// TIA Portal project "Njegovec_diplomski_PLC_HMI" (V19)

(* hardware
DEVICE "S7-1500/ET200MP station_1"  S7-1500 station
   slot 0: "Rail_0"  Rack  6ES7 590-1***0-0AA0
   slot 1: "PLC_1"  CPU 1513-1 PN  6ES7 513-1AL02-0AB0  V2.6
      slot 3: "CPU display_1"  6ES7591-1AA00-0AA0
      slot 32768: "PROFINET interface_1"  X1
DEVICE "HMI_1"  KTP700 Basic PN
   slot 0: "HMI_1"  KTP700 Basic PN  6AV2 123-2GB03-0AX0  17.0.0.0
   slot 1: "HMI_RT_1"  KTP700 Basic PN  6AV2 123-2GB03-0AX0  17.0.0.0
   slot 5: "HMI_1.IE_CP_1"  PROFINET Interface  17.0.0.0
      slot 1: "PROFINET Interface_1"  PROFINET Interface
         slot 1: "Port_1"  Port
*)

// ===== PLC "PLC_1"  CPU 1513-1 PN =====

VAR_GLOBAL   // PLC tag table "Default tag table"
   "air_ON" AT %M4.0 : Bool;
   "System_Byte" AT %MB100 : Byte;
   "FirstScan" AT %M100.0 : Bool;
   "DiagStatusUpdate" AT %M100.1 : Bool;
   "AlwaysTRUE" AT %M100.2 : Bool;
   "AlwaysFALSE" AT %M100.3 : Bool;
   "Clock_Byte" AT %MB105 : Byte;
   "Clock_10Hz" AT %M105.0 : Bool;
   "Clock_5Hz" AT %M105.1 : Bool;
   "Clock_2.5Hz" AT %M105.2 : Bool;
   "Clock_2Hz" AT %M105.3 : Bool;
   "Clock_1.25Hz" AT %M105.4 : Bool;
   "Clock_1Hz" AT %M105.5 : Bool;
   "Clock_0.625Hz" AT %M105.6 : Bool;
   "Clock_0.5Hz" AT %M105.7 : Bool;
END_VAR

VAR_GLOBAL   // PLC tag table "Okretni stol"
   "ventil_1_ukljuci" AT %Q0.1 : Bool;
   "ventil_1_iskljuci" AT %Q0.2 : Bool;
   "stol_okret" AT %Q1.5 : Bool;
   "ventil_2_ukljuci" AT %Q0.3 : Bool;
   "ventil_2_iskljuci" AT %Q0.4 : Bool;
   "clamp_1_1_otvoren" AT %I0.1 : Bool;
   "clamp_2_1_otvoren" AT %I0.3 : Bool;
   "clamp_3_1_otvoren" AT %I0.5 : Bool;
   "clamp_4_1_otvoren" AT %I0.7 : Bool;
   "clamp_5_1_otvoren" AT %I1.1 : Bool;
   "clamp_1_2_otvoren" AT %I1.3 : Bool;
   "clamp_2_2_otvoren" AT %I1.5 : Bool;
   "clamp_3_2_otvoren" AT %I1.7 : Bool;
   "clamp_4_2_otvoren" AT %I2.1 : Bool;
   "clamp_5_2_otvoren" AT %I2.3 : Bool;
   "pin_1_1_izvucen" AT %I2.5 : Bool;
   "pin_2_1_izvucen" AT %I2.7 : Bool;
   "pin_3_1_izvucen" AT %I3.1 : Bool;
   "pin_1_2_izvucen" AT %I3.3 : Bool;
   "pin_2_2_izvucen" AT %I3.5 : Bool;
   "pin_3_2_izvucen" AT %I3.7 : Bool;
   "clamp_1_1_zatvoren" AT %I0.0 : Bool;
   "clamp_2_1_zatvoren" AT %I0.2 : Bool;
   "clamp_3_1_zatvoren" AT %I0.4 : Bool;
   "clamp_4_1_zatvoren" AT %I0.6 : Bool;
   "clamp_5_1_zatvoren" AT %I1.0 : Bool;
   "clamp_1_2_zatvoren" AT %I1.2 : Bool;
   "clamp_2_2_zatvoren" AT %I1.4 : Bool;
   "clamp_3_2_zatvoren" AT %I1.6 : Bool;
   "clamp_4_2_zatvoren" AT %I2.0 : Bool;
   "clamp_5_2_zatvoren" AT %I2.2 : Bool;
   "pin_1_1_uvucen" AT %I2.4 : Bool;
   "pin_2_1_uvucen" AT %I2.6 : Bool;
   "pin_3_1_uvucen" AT %I3.0 : Bool;
   "pin_1_2_uvucen" AT %I3.2 : Bool;
   "pin_2_2_uvucen" AT %I3.4 : Bool;
   "pin_3_2_uvucen" AT %I3.6 : Bool;
   "ventil_pin_1_uklj" AT %Q1.1 : Bool;
   "ventil_pin_1_isklj" AT %Q1.2 : Bool;
   "ventil_pin_2_uklj" AT %Q1.3 : Bool;
   "ventil_pin_2_isklj" AT %Q1.4 : Bool;
   "stol_povratak" AT %Q1.6 : Bool;
   "stol_home" AT %I4.0 : Bool;
   "stol_final" AT %I4.1 : Bool;
END_VAR

VAR_GLOBAL   // PLC tag table "Tipkalo"
   "zeleno" AT %M1.0 : Bool;
   "bijelo" AT %M1.1 : Bool;
   "plavo" AT %M1.2 : Bool;
   "zahtjev_vrata" AT %M1.3 : Bool;
END_VAR

VAR_GLOBAL   // PLC tag table "Robot"
   "robot_move_enable" AT %M2.0 : Bool;
   "KR120_R2700_2_at_HOME" AT %I5.0 : Bool;
   "KR120_R2700_2_startProgram" AT %Q2.0 : Bool;
   "KR120_R2700_2_emergencyStop" AT %Q2.1 : Bool;
   "KR120_R2700_2_programPause" AT %Q2.2 : Bool;
   "KR120_R2700_2_programEnded" AT %I5.1 : Bool;
   "KR120_R2700_2_robotReady" AT %I5.2 : Bool;
   "KR120_R2700_2_mirrorProgramNumber" AT %IB6 : Byte;
   "KR120_R2700_2_programNumber" AT %QB6 : Byte;
   "Zavar_gotov" AT %I8.6 : Bool;
   "handshake_test_out" AT %Q4.0 : Bool;
   "pocetak_rada" AT %I7.1 : Bool;
END_VAR

VAR_GLOBAL   // PLC tag table "Safety"
   "EstopOK" AT %M3.0 : Bool;
END_VAR

VAR_GLOBAL   // PLC tag table "Vrata"
   "vrata_otvori" AT %Q3.0 : Bool;
   "vrata_zatvori" AT %Q3.1 : Bool;
   "lock_zat" AT %Q4.1 : Bool;
   "lock_otv" AT %Q4.2 : Bool;
   "otvoren_lock" AT %I7.0 : Bool;
   "zatvoren_lock" AT %I7.2 : Bool;
   "rolo_vrata_zatvorena" AT %I7.3 : Bool;
   "rolo_vrata_otvorena" AT %I7.4 : Bool;
END_VAR

VAR_GLOBAL   // PLC tag table "Radni_komad"
   "Op2_manji_okvir_start" AT %Q3.2 : Bool;
   "Okvir_manji_unisti_start" AT %Q3.3 : Bool;
   "Op2_manji_okvir_end" AT %I4.6 : Bool;
   "Op3_zavareni_start" AT %Q3.6 : Bool;
   "Zavareno_unisti_start" AT %Q3.7 : Bool;
   "s1_md_prisutan" AT %I4.2 : Bool;
   "s1_vd_prisutan" AT %I4.3 : Bool;
   "s2_md_prisutan" AT %I4.4 : Bool;
   "s2_vd_prisutan" AT %I4.5 : Bool;
   "Op1_veci_okvir_start" AT %Q3.4 : Bool;
   "Okvir_veci_unisti_start" AT %Q3.5 : Bool;
   "Op1_veci_okvir_end" AT %I4.7 : Bool;
   "s1_vk_ind1" AT %I5.4 : Bool;
   "s1_vk_ind2" AT %I5.5 : Bool;
   "s1_mk_ind" AT %I5.6 : Bool;
   "Op3_zavareni_end" AT %I5.7 : Bool;
   "Zavareno_unisti_end" AT %I7.5 : Bool;
   "Op1_veci_okvir_end_2" AT %I8.0 : Bool;
   "Okvir_veci_unisti_end_2" AT %I8.1 : Bool;
   "Op2_manji_okvir_end_2" AT %I8.2 : Bool;
   "Okvir_manji_unisti_end_2" AT %I8.3 : Bool;
   "Op3_zavareni_end_2" AT %I8.4 : Bool;
   "Zavareno_unisti_end_2" AT %I8.5 : Bool;
   "Op1_veci_okvir_2_start" AT %Q7.1 : Bool;
   "Op2_manji_okvir_2_start" AT %Q7.2 : Bool;
   "Op3_zavareni_2_start" AT %Q7.3 : Bool;
   "Okvir_veci_unisti_2_start" AT %Q7.4 : Bool;
   "Zavareno_unisti_2_start" AT %Q7.5 : Bool;
   "Okvir_manji_unisti_2_start" AT %Q7.6 : Bool;
   "s2_vk_ind1" AT %I9.0 : Bool;
   "s2_vk_ind2" AT %I9.1 : Bool;
   "s2_mk_ind" AT %I9.2 : Bool;
END_VAR

VAR_GLOBAL   // PLC tag table "Semafor"
   "zeleno_svjetlo" AT %I5.3 : Bool;
   "zuto_svjetlo" AT %I7.6 : Bool;
   "crveno_svjetlo" AT %I7.7 : Bool;
END_VAR

// folder: Glavni_program

DATA_BLOCK "pom_bits"   // DB1
{ S7_Optimized_Access := 'TRUE' }
VERSION : 0.1
   VAR
      start_auto : Bool;
      automatika_aktivna : Bool;
      iskljucivanje_v_2 : Bool;
      okret : Bool;
      dio_dodan : Bool;
      spremno_za_okret : Bool;
      robot_gotov : Bool;
      sigurnosni_skener_OK : Bool;
      safety_OK : Bool;
   END_VAR
BEGIN
END_DATA_BLOCK

DATA_BLOCK "GlavniProgram_DB"   // DB2
{ S7_Optimized_Access := 'TRUE' }
VERSION : 0.1
// stored: InstanceOfName GlavniProgram
"GlavniProgram"
BEGIN
END_DATA_BLOCK

DATA_BLOCK "Handshake"   // DB10
{ S7_Optimized_Access := 'TRUE' }
VERSION : 0.1
   VAR
      Stol_PLC : Bool;
      Spremna_opskrba : Bool;
      Stol_PLC_OK : Bool;
      Spremno_za_stez_i_okret : Bool;
      Spremno_za_stez_i_povrat : Bool;
      Spremno_za_varenje : Bool;
   END_VAR
BEGIN
END_DATA_BLOCK

// folder: HMI

DATA_BLOCK "Errors"   // DB3
{ S7_Optimized_Access := 'TRUE' }
VERSION : 0.1
   VAR
      error_bit : Bool;
      err_zrak : Bool;
      err_Estop : Bool;
      err_raspored : Bool;
      err_vrata_otvorena : Bool;
   END_VAR
BEGIN
END_DATA_BLOCK

DATA_BLOCK "HMI_signals"   // DB7
{ S7_Optimized_Access := 'TRUE' }
VERSION : 0.1
   VAR
      setup_mode : Bool;
      auto_mode : Bool;
      robot_start : Bool;
      robot_stop : Bool;
      robot_em_stop : Bool;
      set_ventil1_ukljuci : Bool;
      set_ventil1_iskljuci : Bool;
      set_ventil2_ukljuci : Bool;
      set_ventil2_iskljuci : Bool;
      set_okret : Bool;
      set_povratak : Bool;
      set_vrata_otvori : Bool;
      set_vrata_zatvori : Bool;
      set_ventil1_pin_ukljuci : Bool;
      set_ventil1_pin_iskljuci : Bool;
      set_ventil2_pin_ukljuci : Bool;
      set_ventil2_pin_iskljuci : Bool;
      s1_md_prisutan : Bool;
      s1_vd_prisutan : Bool;
      set_s1_md_stvori : Bool;
      set_s1_md_unisti : Bool;
      set_s1_vd_stvori : Bool;
      set_s1_vd_unisti : Bool;
      set_s1_md_stvori_2 : Bool;
      set_s1_md_unisti_2 : Bool;
      set_s1_vd_stvori_2 : Bool;
      set_s1_vd_unisti_2 : Bool;
      set_zavareni : Bool;
      set_zavareni_2 : Bool;
      prog_zavar : Bool;
      prog_brusenje : Bool;
      sek_stol_res : Bool;
      sek_rob_res : Bool;
      sek_glav_res : Bool;
      strana_1_prisutni : Bool;
      strana_2_prisutni : Bool;
      set_unisti_zavarene : Bool;
      set_unisti_zavarene_2 : Bool;
      lock_otv : Bool;
      lock_zat : Bool;
      zahtjev_za_vrata : Bool;
      zrak_u_sustavu : Bool;
      set_zrak : Bool;
      reset_zrak : Bool;
      Estop : Bool := true;
   END_VAR
BEGIN
END_DATA_BLOCK

// folder: Sekvence

DATA_BLOCK "Sekvence_DB"   // DB11
{ S7_Optimized_Access := 'TRUE' }
VERSION : 0.1
   VAR
      vrata_otvori : Bool;
      vrata_zatvori : Bool;
      Zavareno_unisti_start : Bool;
      Zavareno_unisti_2_start : Bool;
      ventil_1_iskljuci : Bool;
      ventil_1_ukljuci : Bool;
      ventil_pin_1_uklj : Bool;
      ventil_pin_1_isklj : Bool;
      stol_okret : Bool;
      ventil_2_ukljuci : Bool;
      ventil_2_iskljuci : Bool;
      ventil_pin_2_uklj : Bool;
      ventil_pin_2_isklj : Bool;
      stol_povratak : Bool;
      KR120_R2700_2_startProgram : Bool;
      KR120_R2700_2_emergencyStop : Bool;
      KR120_R2700_2_programPause : Bool;
      Op2_manji_okvir_start : Bool;
      Okvir_manji_unisti_start : Bool;
      Op1_veci_okvir_start : Bool;
      Okvir_veci_unisti_start : Bool;
      Op3_zavareni_start : Bool;
      lock_zat : Bool;
      lock_otv : Bool;
      KR120_R2700_2_programNumber : Byte;
      Op2_manji_okvir_2_start : Bool;
      Op1_veci_okvir_2_start : Bool;
      Op3_zavareni_2_start : Bool;
   END_VAR
BEGIN
END_DATA_BLOCK

DATA_BLOCK "Glavna_sekvenca_DB"   // DB12
{ S7_Optimized_Access := 'TRUE' }
VERSION : 0.1
// stored: InstanceOfName Glavna_sekvenca
"Glavna_sekvenca"
BEGIN
END_DATA_BLOCK

DATA_BLOCK "Okretni_stol_sekvenca_DB"   // DB13
{ S7_Optimized_Access := 'TRUE' }
VERSION : 0.1
// stored: InstanceOfName Okretni_stol_sekvenca
"Okretni_stol_sekvenca"
BEGIN
END_DATA_BLOCK

DATA_BLOCK "Robot_sekvenca_DB"   // DB14
{ S7_Optimized_Access := 'TRUE' }
VERSION : 0.1
// stored: InstanceOfName Robot_sekvenca
"Robot_sekvenca"
BEGIN
END_DATA_BLOCK

// folder: Senzori

DATA_BLOCK "Senzori"   // DB4
{ S7_Optimized_Access := 'TRUE' }
VERSION : 0.1
   VAR
      clamps1_open : Bool;
      clamps2_open : Bool;
      clamps1_closed : Bool;
      clamps2_closed : Bool;
      pins1_out : Bool;
      pins1_in : Bool;
      pins2_out : Bool;
      pins2_in : Bool;
   END_VAR
BEGIN
END_DATA_BLOCK

DATA_BLOCK "Senzori_prog_DB"   // DB8
{ S7_Optimized_Access := 'TRUE' }
VERSION : 0.1
// stored: InstanceOfName Senzori_prog
"Senzori_prog"
BEGIN
END_DATA_BLOCK

// folder: System blocks/Program resources

DATA_BLOCK "err_timer"   // DB5
{ S7_Optimized_Access := 'TRUE' }
AUTHOR : Simatic
FAMILY : IEC
NAME : IEC_TMR
VERSION : 1.0
// stored: InstanceOfName IEC_TIMER
"IEC_TIMER"
BEGIN
END_DATA_BLOCK

DATA_BLOCK "IEC_Timer_0_DB"   // DB9
{ S7_Optimized_Access := 'TRUE' }
AUTHOR : Simatic
FAMILY : IEC
NAME : IEC_TMR
VERSION : 1.0
// stored: InstanceOfName IEC_TIMER
"IEC_TIMER"
BEGIN
END_DATA_BLOCK

// folder: (top level)

ORGANIZATION_BLOCK "Main"   // OB1, LAD, ProgramCycle
TITLE = "Main Program Sweep (Cycle)"
{ S7_Optimized_Access := 'TRUE' }
VERSION : 0.1
   VAR_INPUT
      Initial_Call : Bool;   // Initial call of this OB
      Remanence : Bool;   // =True, if remanent data are available
   END_VAR
BEGIN

REGION Network 1: Pozivi blokova
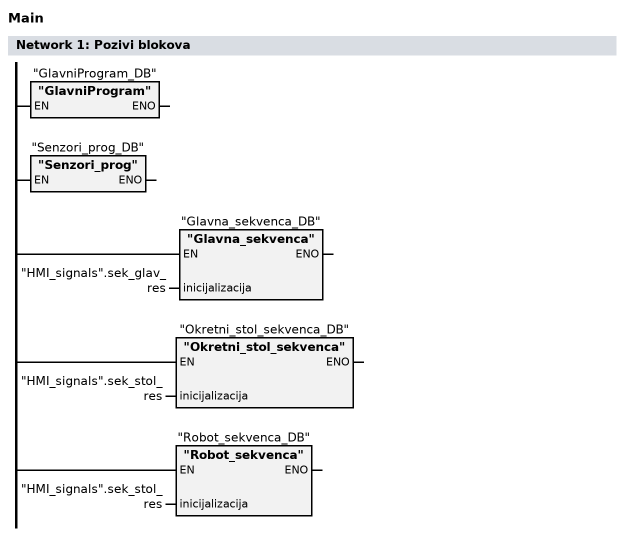
   RUNG wire#powerrail
      "GlavniProgram_DB"()
   END_RUNG
   RUNG wire#powerrail
      "Senzori_prog_DB"()
   END_RUNG
   RUNG wire#powerrail
      "Glavna_sekvenca_DB"(inicijalizacija := "HMI_signals".sek_glav_res)
   END_RUNG
   RUNG wire#powerrail
      "Okretni_stol_sekvenca_DB"(inicijalizacija := "HMI_signals".sek_stol_res)
   END_RUNG
   RUNG wire#powerrail
      "Robot_sekvenca_DB"(inicijalizacija := "HMI_signals".sek_stol_res)
   END_RUNG
   // the same network as SCL:
   "GlavniProgram_DB"();   // "GlavniProgram"
   "Senzori_prog_DB"();   // "Senzori_prog"
   "Glavna_sekvenca_DB"(inicijalizacija := "HMI_signals".sek_glav_res);   // "Glavna_sekvenca"
   "Okretni_stol_sekvenca_DB"(inicijalizacija := "HMI_signals".sek_stol_res);   // "Okretni_stol_sekvenca"
   "Robot_sekvenca_DB"(inicijalizacija := "HMI_signals".sek_stol_res);   // "Robot_sekvenca"
END_REGION
END_ORGANIZATION_BLOCK

// folder: Glavni_program

FUNCTION_BLOCK "GlavniProgram"   // FB1, LAD
{ S7_Optimized_Access := 'TRUE' }
VERSION : 0.1
   VAR
      pom_stol_okrenut : Bool;
      stepNum : Int;
      safety_OK : Bool;
      bit_na_brid : Array[0..12] of Bool;
      zahtjev_poslan : Bool;
   END_VAR
   VAR_TEMP   // added for the SCL form of the ladder/FBD networks
      _w1 : Bool;
      _w2 : Bool;
      _w3 : Bool;
      _w4 : Bool;
      _w5 : Bool;
      _w6 : Bool;
   END_VAR
BEGIN

REGION Network 1: Pokretanje i prekidanje automatskog načina rada
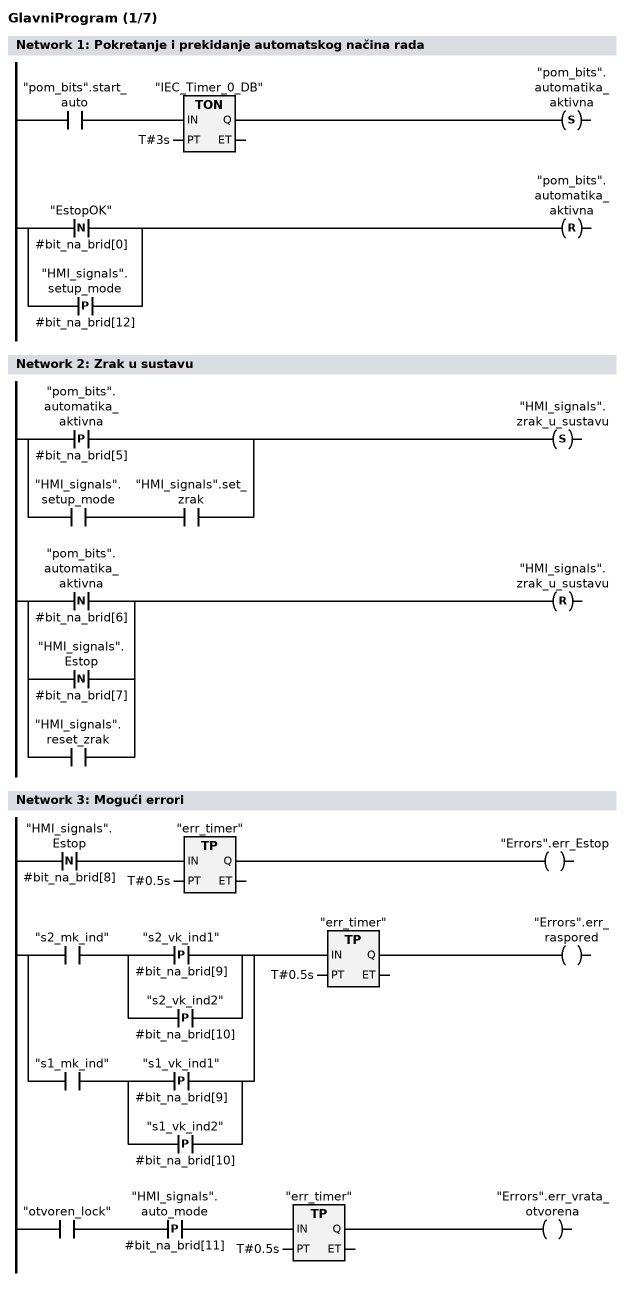
   "IEC_Timer_0_DB".TON(IN := "pom_bits".start_auto, PT := T#3s);
   IF "IEC_Timer_0_DB".Q THEN "pom_bits".automatika_aktivna := TRUE; END_IF;
   #_w1 := NOT "EstopOK" AND #bit_na_brid[0];   // falling edge of "EstopOK"
   #bit_na_brid[0] := "EstopOK";
   #_w2 := "HMI_signals".setup_mode AND NOT #bit_na_brid[12];   // rising edge of "HMI_signals".setup_mode
   #bit_na_brid[12] := "HMI_signals".setup_mode;
   IF #_w1 OR #_w2 THEN "pom_bits".automatika_aktivna := FALSE; END_IF;
END_REGION

REGION Network 2: Zrak u sustavu
   RUNG wire#powerrail
      P_Contact(operand := "pom_bits".automatika_aktivna, bit := #bit_na_brid[5])
      wire#w1
      S_Coil( "HMI_signals".zrak_u_sustavu )
   END_RUNG
   RUNG wire#powerrail
      Contact( "HMI_signals".setup_mode )
      Contact( "HMI_signals".set_zrak )
   END_RUNG wire#w1
   RUNG wire#powerrail
      N_Contact(operand := "pom_bits".automatika_aktivna, bit := #bit_na_brid[6])
      wire#w2
      R_Coil( "HMI_signals".zrak_u_sustavu )
   END_RUNG
   RUNG wire#powerrail
      N_Contact(operand := "HMI_signals".Estop, bit := #bit_na_brid[7])
   END_RUNG wire#w2
   RUNG wire#powerrail
      Contact( "HMI_signals".reset_zrak )
   END_RUNG wire#w2
   // the same network as SCL:
   #_w1 := "pom_bits".automatika_aktivna AND NOT #bit_na_brid[5];   // rising edge of "pom_bits".automatika_aktivna
   #bit_na_brid[5] := "pom_bits".automatika_aktivna;
   IF #_w1 OR ("HMI_signals".setup_mode AND "HMI_signals".set_zrak) THEN
       "HMI_signals".zrak_u_sustavu := TRUE;
   END_IF;
   #_w2 := NOT "pom_bits".automatika_aktivna AND #bit_na_brid[6];   // falling edge of "pom_bits".automatika_aktivna
   #bit_na_brid[6] := "pom_bits".automatika_aktivna;
   #_w3 := NOT "HMI_signals".Estop AND #bit_na_brid[7];   // falling edge of "HMI_signals".Estop
   #bit_na_brid[7] := "HMI_signals".Estop;
   IF #_w2 OR #_w3 OR "HMI_signals".reset_zrak THEN "HMI_signals".zrak_u_sustavu := FALSE; END_IF;
END_REGION

REGION Network 3: Mogući errori
   #_w1 := NOT "HMI_signals".Estop AND #bit_na_brid[8];   // falling edge of "HMI_signals".Estop
   #bit_na_brid[8] := "HMI_signals".Estop;
   "err_timer".TP(IN := #_w1, PT := T#0.5s);
   "Errors".err_Estop := "err_timer".Q;
   #_w2 := "s2_mk_ind" AND "s2_vk_ind1" AND NOT #bit_na_brid[9];   // rising edge of "s2_vk_ind1"
   #bit_na_brid[9] := "s2_vk_ind1";
   #_w3 := "s2_mk_ind" AND "s2_vk_ind2" AND NOT #bit_na_brid[10];   // rising edge of "s2_vk_ind2"
   #bit_na_brid[10] := "s2_vk_ind2";
   #_w4 := "s1_mk_ind" AND "s1_vk_ind1" AND NOT #bit_na_brid[9];   // rising edge of "s1_vk_ind1"
   #bit_na_brid[9] := "s1_vk_ind1";
   #_w5 := "s1_mk_ind" AND "s1_vk_ind2" AND NOT #bit_na_brid[10];   // rising edge of "s1_vk_ind2"
   #bit_na_brid[10] := "s1_vk_ind2";
   "err_timer".TP(IN := #_w2 OR #_w3 OR #_w4 OR #_w5, PT := T#0.5s);
   "Errors".err_raspored := "err_timer".Q;
   #_w6 := "otvoren_lock" AND "HMI_signals".auto_mode AND NOT #bit_na_brid[11];   // rising edge of "HMI_signals".auto_mode
   #bit_na_brid[11] := "HMI_signals".auto_mode;
   "err_timer".TP(IN := #_w6, PT := T#0.5s);
   "Errors".err_vrata_otvorena := "err_timer".Q;
END_REGION

REGION Network 4: Aktivacija error bita
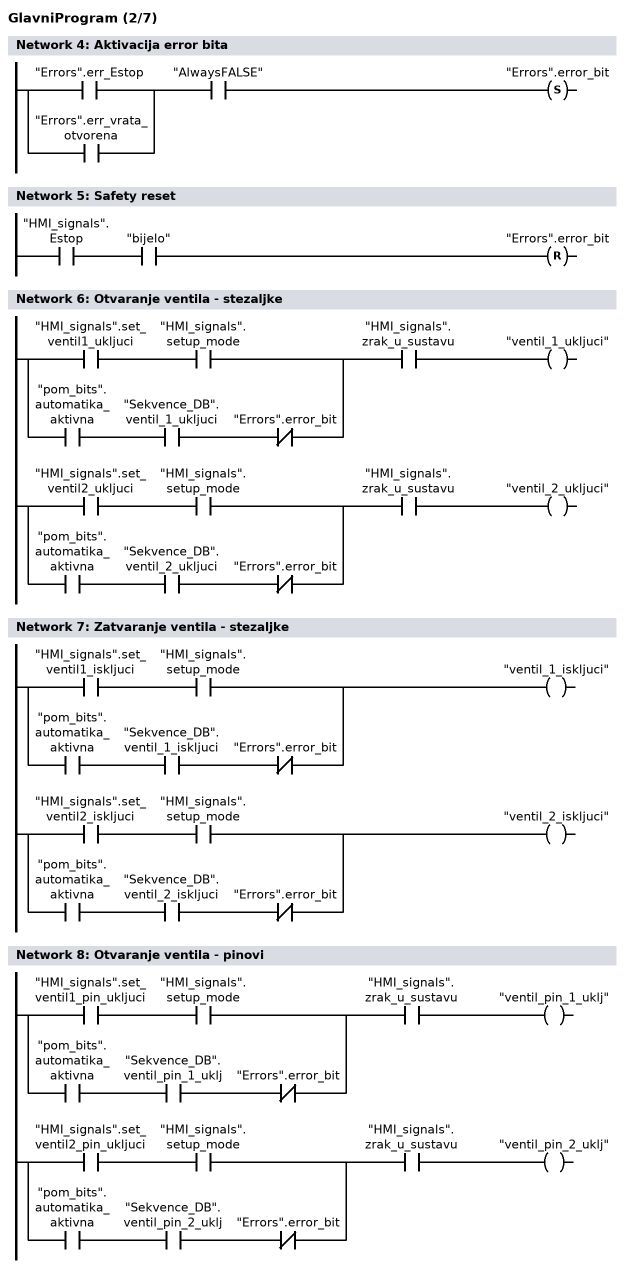
   RUNG wire#powerrail
      Contact( "Errors".err_Estop )
      wire#w1
      Contact( "AlwaysFALSE" )
      S_Coil( "Errors".error_bit )
   END_RUNG
   RUNG wire#powerrail
      Contact( "Errors".err_vrata_otvorena )
   END_RUNG wire#w1
   // the same network as SCL:
   IF ("Errors".err_Estop OR "Errors".err_vrata_otvorena) AND "AlwaysFALSE" THEN
       "Errors".error_bit := TRUE;
   END_IF;
END_REGION

REGION Network 5: Safety reset
   RUNG wire#powerrail
      Contact( "HMI_signals".Estop )
      Contact( "bijelo" )
      R_Coil( "Errors".error_bit )
   END_RUNG
   // the same network as SCL:
   IF "HMI_signals".Estop AND "bijelo" THEN "Errors".error_bit := FALSE; END_IF;
END_REGION

REGION Network 6: Otvaranje ventila - stezaljke
   RUNG wire#powerrail
      Contact( "HMI_signals".set_ventil1_ukljuci )
      Contact( "HMI_signals".setup_mode )
      wire#w1
      Contact( "HMI_signals".zrak_u_sustavu )
      Coil( "ventil_1_ukljuci" )
   END_RUNG
   RUNG wire#powerrail
      Contact( "pom_bits".automatika_aktivna )
      Contact( "Sekvence_DB".ventil_1_ukljuci )
      I_Contact( "Errors".error_bit )
   END_RUNG wire#w1
   RUNG wire#powerrail
      Contact( "HMI_signals".set_ventil2_ukljuci )
      Contact( "HMI_signals".setup_mode )
      wire#w2
      Contact( "HMI_signals".zrak_u_sustavu )
      Coil( "ventil_2_ukljuci" )
   END_RUNG
   RUNG wire#powerrail
      Contact( "pom_bits".automatika_aktivna )
      Contact( "Sekvence_DB".ventil_2_ukljuci )
      I_Contact( "Errors".error_bit )
   END_RUNG wire#w2
   // the same network as SCL:
   "ventil_1_ukljuci" := (("HMI_signals".set_ventil1_ukljuci AND "HMI_signals".setup_mode) OR ("pom_bits".automatika_aktivna AND "Sekvence_DB".ventil_1_ukljuci AND NOT "Errors".error_bit)) AND "HMI_signals".zrak_u_sustavu;
   "ventil_2_ukljuci" := (("HMI_signals".set_ventil2_ukljuci AND "HMI_signals".setup_mode) OR ("pom_bits".automatika_aktivna AND "Sekvence_DB".ventil_2_ukljuci AND NOT "Errors".error_bit)) AND "HMI_signals".zrak_u_sustavu;
END_REGION

REGION Network 7: Zatvaranje ventila - stezaljke
   RUNG wire#powerrail
      Contact( "HMI_signals".set_ventil1_iskljuci )
      Contact( "HMI_signals".setup_mode )
      wire#w1
      Coil( "ventil_1_iskljuci" )
   END_RUNG
   RUNG wire#powerrail
      Contact( "pom_bits".automatika_aktivna )
      Contact( "Sekvence_DB".ventil_1_iskljuci )
      I_Contact( "Errors".error_bit )
   END_RUNG wire#w1
   RUNG wire#powerrail
      Contact( "HMI_signals".set_ventil2_iskljuci )
      Contact( "HMI_signals".setup_mode )
      wire#w2
      Coil( "ventil_2_iskljuci" )
   END_RUNG
   RUNG wire#powerrail
      Contact( "pom_bits".automatika_aktivna )
      Contact( "Sekvence_DB".ventil_2_iskljuci )
      I_Contact( "Errors".error_bit )
   END_RUNG wire#w2
   // the same network as SCL:
   "ventil_1_iskljuci" := ("HMI_signals".set_ventil1_iskljuci AND "HMI_signals".setup_mode) OR ("pom_bits".automatika_aktivna AND "Sekvence_DB".ventil_1_iskljuci AND NOT "Errors".error_bit);
   "ventil_2_iskljuci" := ("HMI_signals".set_ventil2_iskljuci AND "HMI_signals".setup_mode) OR ("pom_bits".automatika_aktivna AND "Sekvence_DB".ventil_2_iskljuci AND NOT "Errors".error_bit);
END_REGION

REGION Network 8: Otvaranje ventila - pinovi
   RUNG wire#powerrail
      Contact( "HMI_signals".set_ventil1_pin_ukljuci )
      Contact( "HMI_signals".setup_mode )
      wire#w1
      Contact( "HMI_signals".zrak_u_sustavu )
      Coil( "ventil_pin_1_uklj" )
   END_RUNG
   RUNG wire#powerrail
      Contact( "pom_bits".automatika_aktivna )
      Contact( "Sekvence_DB".ventil_pin_1_uklj )
      I_Contact( "Errors".error_bit )
   END_RUNG wire#w1
   RUNG wire#powerrail
      Contact( "HMI_signals".set_ventil2_pin_ukljuci )
      Contact( "HMI_signals".setup_mode )
      wire#w2
      Contact( "HMI_signals".zrak_u_sustavu )
      Coil( "ventil_pin_2_uklj" )
   END_RUNG
   RUNG wire#powerrail
      Contact( "pom_bits".automatika_aktivna )
      Contact( "Sekvence_DB".ventil_pin_2_uklj )
      I_Contact( "Errors".error_bit )
   END_RUNG wire#w2
   // the same network as SCL:
   "ventil_pin_1_uklj" := (("HMI_signals".set_ventil1_pin_ukljuci AND "HMI_signals".setup_mode) OR ("pom_bits".automatika_aktivna AND "Sekvence_DB".ventil_pin_1_uklj AND NOT "Errors".error_bit)) AND "HMI_signals".zrak_u_sustavu;
   "ventil_pin_2_uklj" := (("HMI_signals".set_ventil2_pin_ukljuci AND "HMI_signals".setup_mode) OR ("pom_bits".automatika_aktivna AND "Sekvence_DB".ventil_pin_2_uklj AND NOT "Errors".error_bit)) AND "HMI_signals".zrak_u_sustavu;
END_REGION

REGION Network 9: Zatvaranje ventila - pinovi
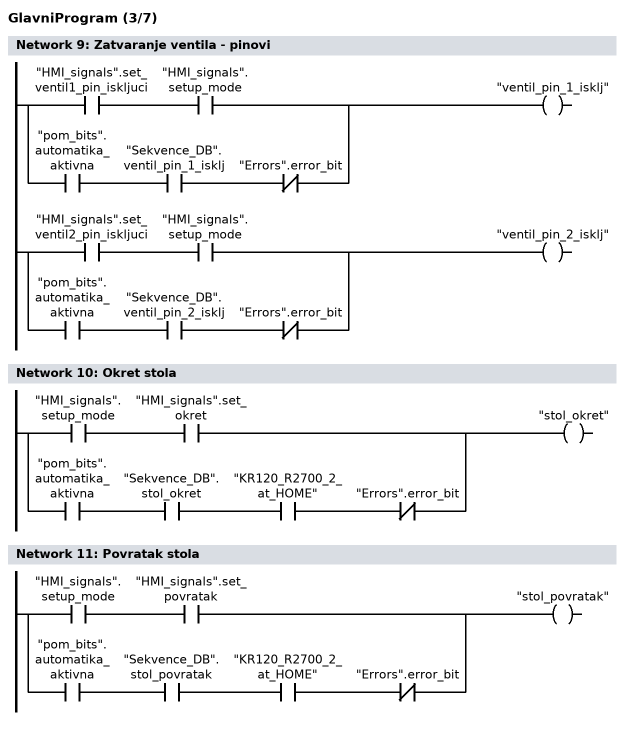
   RUNG wire#powerrail
      Contact( "HMI_signals".set_ventil1_pin_iskljuci )
      Contact( "HMI_signals".setup_mode )
      wire#w1
      Coil( "ventil_pin_1_isklj" )
   END_RUNG
   RUNG wire#powerrail
      Contact( "pom_bits".automatika_aktivna )
      Contact( "Sekvence_DB".ventil_pin_1_isklj )
      I_Contact( "Errors".error_bit )
   END_RUNG wire#w1
   RUNG wire#powerrail
      Contact( "HMI_signals".set_ventil2_pin_iskljuci )
      Contact( "HMI_signals".setup_mode )
      wire#w2
      Coil( "ventil_pin_2_isklj" )
   END_RUNG
   RUNG wire#powerrail
      Contact( "pom_bits".automatika_aktivna )
      Contact( "Sekvence_DB".ventil_pin_2_isklj )
      I_Contact( "Errors".error_bit )
   END_RUNG wire#w2
   // the same network as SCL:
   "ventil_pin_1_isklj" := ("HMI_signals".set_ventil1_pin_iskljuci AND "HMI_signals".setup_mode) OR ("pom_bits".automatika_aktivna AND "Sekvence_DB".ventil_pin_1_isklj AND NOT "Errors".error_bit);
   "ventil_pin_2_isklj" := ("HMI_signals".set_ventil2_pin_iskljuci AND "HMI_signals".setup_mode) OR ("pom_bits".automatika_aktivna AND "Sekvence_DB".ventil_pin_2_isklj AND NOT "Errors".error_bit);
END_REGION

REGION Network 10: Okret stola
   RUNG wire#powerrail
      Contact( "HMI_signals".setup_mode )
      Contact( "HMI_signals".set_okret )
      wire#w1
      Coil( "stol_okret" )
   END_RUNG
   RUNG wire#powerrail
      Contact( "pom_bits".automatika_aktivna )
      Contact( "Sekvence_DB".stol_okret )
      Contact( "KR120_R2700_2_at_HOME" )
      I_Contact( "Errors".error_bit )
   END_RUNG wire#w1
   // the same network as SCL:
   "stol_okret" := ("HMI_signals".setup_mode AND "HMI_signals".set_okret) OR ("pom_bits".automatika_aktivna AND "Sekvence_DB".stol_okret AND "KR120_R2700_2_at_HOME" AND NOT "Errors".error_bit);
END_REGION

REGION Network 11: Povratak stola
   RUNG wire#powerrail
      Contact( "HMI_signals".setup_mode )
      Contact( "HMI_signals".set_povratak )
      wire#w1
      Coil( "stol_povratak" )
   END_RUNG
   RUNG wire#powerrail
      Contact( "pom_bits".automatika_aktivna )
      Contact( "Sekvence_DB".stol_povratak )
      Contact( "KR120_R2700_2_at_HOME" )
      I_Contact( "Errors".error_bit )
   END_RUNG wire#w1
   // the same network as SCL:
   "stol_povratak" := ("HMI_signals".setup_mode AND "HMI_signals".set_povratak) OR ("pom_bits".automatika_aktivna AND "Sekvence_DB".stol_povratak AND "KR120_R2700_2_at_HOME" AND NOT "Errors".error_bit);
END_REGION

REGION Network 12: Robot
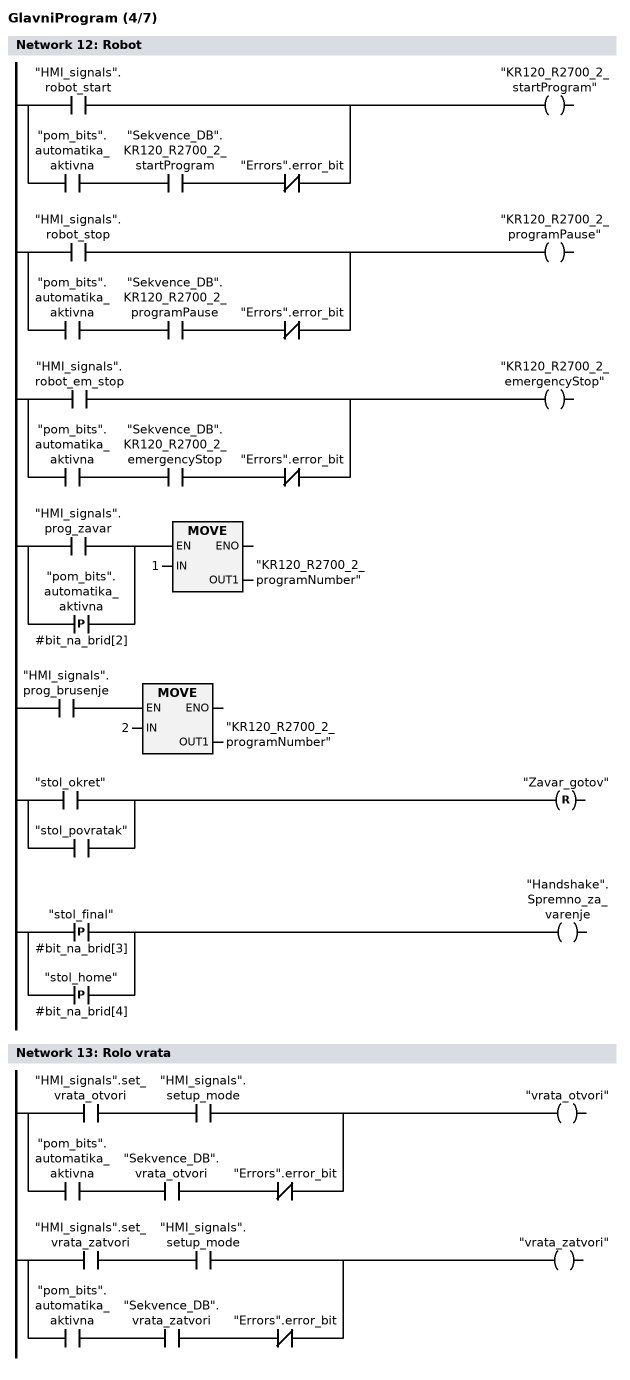
   RUNG wire#powerrail
      Contact( "HMI_signals".robot_start )
      wire#w1
      Coil( "KR120_R2700_2_startProgram" )
   END_RUNG
   RUNG wire#powerrail
      Contact( "pom_bits".automatika_aktivna )
      Contact( "Sekvence_DB".KR120_R2700_2_startProgram )
      I_Contact( "Errors".error_bit )
   END_RUNG wire#w1
   RUNG wire#powerrail
      Contact( "HMI_signals".robot_stop )
      wire#w2
      Coil( "KR120_R2700_2_programPause" )
   END_RUNG
   RUNG wire#powerrail
      Contact( "pom_bits".automatika_aktivna )
      Contact( "Sekvence_DB".KR120_R2700_2_programPause )
      I_Contact( "Errors".error_bit )
   END_RUNG wire#w2
   RUNG wire#powerrail
      Contact( "HMI_signals".robot_em_stop )
      wire#w3
      Coil( "KR120_R2700_2_emergencyStop" )
   END_RUNG
   RUNG wire#powerrail
      Contact( "pom_bits".automatika_aktivna )
      Contact( "Sekvence_DB".KR120_R2700_2_emergencyStop )
      I_Contact( "Errors".error_bit )
   END_RUNG wire#w3
   RUNG wire#powerrail
      Contact( "HMI_signals".prog_zavar )
      wire#w4
      Move(in := 1, out1 => "KR120_R2700_2_programNumber")
   END_RUNG
   RUNG wire#powerrail
      P_Contact(operand := "pom_bits".automatika_aktivna, bit := #bit_na_brid[2])
   END_RUNG wire#w4
   RUNG wire#powerrail
      Contact( "HMI_signals".prog_brusenje )
      Move(in := 2, out1 => "KR120_R2700_2_programNumber")
   END_RUNG
   RUNG wire#powerrail
      Contact( "stol_okret" )
      wire#w5
      R_Coil( "Zavar_gotov" )
   END_RUNG
   RUNG wire#powerrail
      Contact( "stol_povratak" )
   END_RUNG wire#w5
   RUNG wire#powerrail
      P_Contact(operand := "stol_final", bit := #bit_na_brid[3])
      wire#w6
      Coil( "Handshake".Spremno_za_varenje )
   END_RUNG
   RUNG wire#powerrail
      P_Contact(operand := "stol_home", bit := #bit_na_brid[4])
   END_RUNG wire#w6
   // the same network as SCL:
   "KR120_R2700_2_startProgram" := "HMI_signals".robot_start OR ("pom_bits".automatika_aktivna AND "Sekvence_DB".KR120_R2700_2_startProgram AND NOT "Errors".error_bit);
   "KR120_R2700_2_programPause" := "HMI_signals".robot_stop OR ("pom_bits".automatika_aktivna AND "Sekvence_DB".KR120_R2700_2_programPause AND NOT "Errors".error_bit);
   "KR120_R2700_2_emergencyStop" := "HMI_signals".robot_em_stop OR ("pom_bits".automatika_aktivna AND "Sekvence_DB".KR120_R2700_2_emergencyStop AND NOT "Errors".error_bit);
   #_w1 := "pom_bits".automatika_aktivna AND NOT #bit_na_brid[2];   // rising edge of "pom_bits".automatika_aktivna
   #bit_na_brid[2] := "pom_bits".automatika_aktivna;
   IF "HMI_signals".prog_zavar OR #_w1 THEN "KR120_R2700_2_programNumber" := 1; END_IF;
   IF "HMI_signals".prog_brusenje THEN "KR120_R2700_2_programNumber" := 2; END_IF;
   IF "stol_okret" OR "stol_povratak" THEN "Zavar_gotov" := FALSE; END_IF;
   #_w2 := "stol_final" AND NOT #bit_na_brid[3];   // rising edge of "stol_final"
   #bit_na_brid[3] := "stol_final";
   #_w3 := "stol_home" AND NOT #bit_na_brid[4];   // rising edge of "stol_home"
   #bit_na_brid[4] := "stol_home";
   "Handshake".Spremno_za_varenje := #_w2 OR #_w3;
END_REGION

REGION Network 13: Rolo vrata
   RUNG wire#powerrail
      Contact( "HMI_signals".set_vrata_otvori )
      Contact( "HMI_signals".setup_mode )
      wire#w1
      Coil( "vrata_otvori" )
   END_RUNG
   RUNG wire#powerrail
      Contact( "pom_bits".automatika_aktivna )
      Contact( "Sekvence_DB".vrata_otvori )
      I_Contact( "Errors".error_bit )
   END_RUNG wire#w1
   RUNG wire#powerrail
      Contact( "HMI_signals".set_vrata_zatvori )
      Contact( "HMI_signals".setup_mode )
      wire#w2
      Coil( "vrata_zatvori" )
   END_RUNG
   RUNG wire#powerrail
      Contact( "pom_bits".automatika_aktivna )
      Contact( "Sekvence_DB".vrata_zatvori )
      I_Contact( "Errors".error_bit )
   END_RUNG wire#w2
   // the same network as SCL:
   "vrata_otvori" := ("HMI_signals".set_vrata_otvori AND "HMI_signals".setup_mode) OR ("pom_bits".automatika_aktivna AND "Sekvence_DB".vrata_otvori AND NOT "Errors".error_bit);
   "vrata_zatvori" := ("HMI_signals".set_vrata_zatvori AND "HMI_signals".setup_mode) OR ("pom_bits".automatika_aktivna AND "Sekvence_DB".vrata_zatvori AND NOT "Errors".error_bit);
END_REGION

REGION Network 14: Safety lock vrata
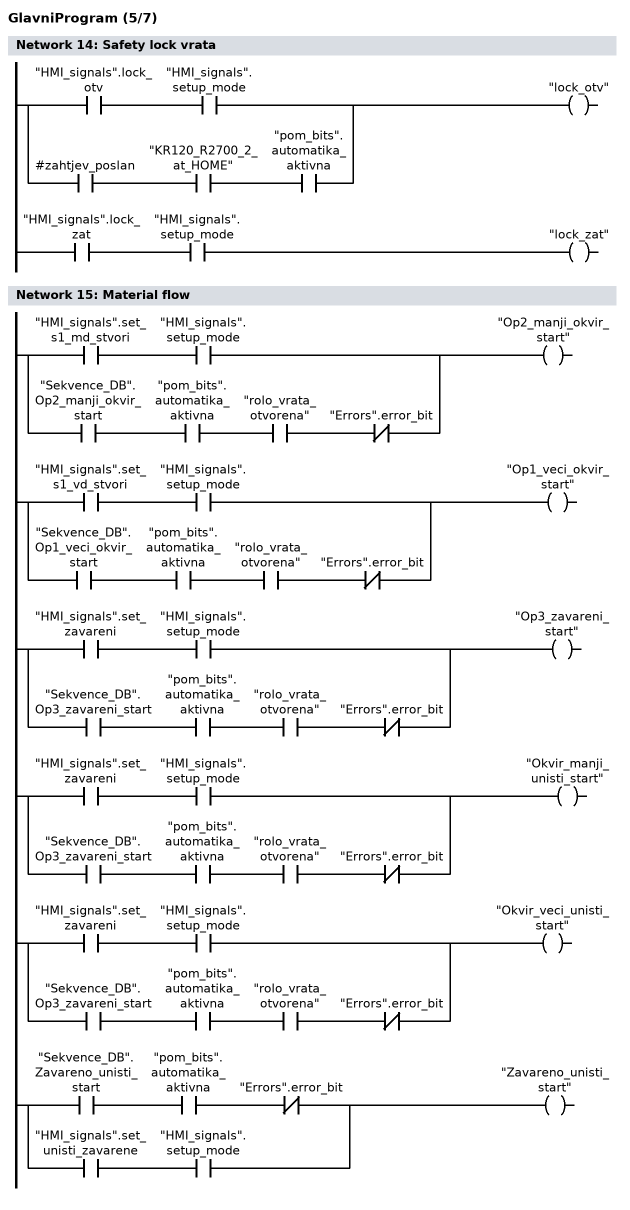
   RUNG wire#powerrail
      Contact( "HMI_signals".lock_otv )
      Contact( "HMI_signals".setup_mode )
      wire#w1
      Coil( "lock_otv" )
   END_RUNG
   RUNG wire#powerrail
      Contact( #zahtjev_poslan )
      Contact( "KR120_R2700_2_at_HOME" )
      Contact( "pom_bits".automatika_aktivna )
   END_RUNG wire#w1
   RUNG wire#powerrail
      Contact( "HMI_signals".lock_zat )
      Contact( "HMI_signals".setup_mode )
      Coil( "lock_zat" )
   END_RUNG
   // the same network as SCL:
   "lock_otv" := ("HMI_signals".lock_otv AND "HMI_signals".setup_mode) OR (#zahtjev_poslan AND "KR120_R2700_2_at_HOME" AND "pom_bits".automatika_aktivna);
   "lock_zat" := "HMI_signals".lock_zat AND "HMI_signals".setup_mode;
END_REGION

REGION Network 15: Material flow
   RUNG wire#powerrail
      Contact( "HMI_signals".set_s1_md_stvori )
      Contact( "HMI_signals".setup_mode )
      wire#w1
      Coil( "Op2_manji_okvir_start" )
   END_RUNG
   RUNG wire#powerrail
      Contact( "Sekvence_DB".Op2_manji_okvir_start )
      Contact( "pom_bits".automatika_aktivna )
      Contact( "rolo_vrata_otvorena" )
      I_Contact( "Errors".error_bit )
   END_RUNG wire#w1
   RUNG wire#powerrail
      Contact( "HMI_signals".set_s1_vd_stvori )
      Contact( "HMI_signals".setup_mode )
      wire#w2
      Coil( "Op1_veci_okvir_start" )
   END_RUNG
   RUNG wire#powerrail
      Contact( "Sekvence_DB".Op1_veci_okvir_start )
      Contact( "pom_bits".automatika_aktivna )
      Contact( "rolo_vrata_otvorena" )
      I_Contact( "Errors".error_bit )
   END_RUNG wire#w2
   RUNG wire#powerrail
      Contact( "HMI_signals".set_zavareni )
      Contact( "HMI_signals".setup_mode )
      wire#w3
      Coil( "Op3_zavareni_start" )
   END_RUNG
   RUNG wire#powerrail
      Contact( "Sekvence_DB".Op3_zavareni_start )
      Contact( "pom_bits".automatika_aktivna )
      Contact( "rolo_vrata_otvorena" )
      I_Contact( "Errors".error_bit )
   END_RUNG wire#w3
   RUNG wire#powerrail
      Contact( "HMI_signals".set_zavareni )
      Contact( "HMI_signals".setup_mode )
      wire#w4
      Coil( "Okvir_manji_unisti_start" )
   END_RUNG
   RUNG wire#powerrail
      Contact( "Sekvence_DB".Op3_zavareni_start )
      Contact( "pom_bits".automatika_aktivna )
      Contact( "rolo_vrata_otvorena" )
      I_Contact( "Errors".error_bit )
   END_RUNG wire#w4
   RUNG wire#powerrail
      Contact( "HMI_signals".set_zavareni )
      Contact( "HMI_signals".setup_mode )
      wire#w5
      Coil( "Okvir_veci_unisti_start" )
   END_RUNG
   RUNG wire#powerrail
      Contact( "Sekvence_DB".Op3_zavareni_start )
      Contact( "pom_bits".automatika_aktivna )
      Contact( "rolo_vrata_otvorena" )
      I_Contact( "Errors".error_bit )
   END_RUNG wire#w5
   RUNG wire#powerrail
      Contact( "Sekvence_DB".Zavareno_unisti_start )
      Contact( "pom_bits".automatika_aktivna )
      I_Contact( "Errors".error_bit )
      wire#w6
      Coil( "Zavareno_unisti_start" )
   END_RUNG
   RUNG wire#powerrail
      Contact( "HMI_signals".set_unisti_zavarene )
      Contact( "HMI_signals".setup_mode )
   END_RUNG wire#w6
   // the same network as SCL:
   "Op2_manji_okvir_start" := ("HMI_signals".set_s1_md_stvori AND "HMI_signals".setup_mode) OR ("Sekvence_DB".Op2_manji_okvir_start AND "pom_bits".automatika_aktivna AND "rolo_vrata_otvorena" AND NOT "Errors".error_bit);
   "Op1_veci_okvir_start" := ("HMI_signals".set_s1_vd_stvori AND "HMI_signals".setup_mode) OR ("Sekvence_DB".Op1_veci_okvir_start AND "pom_bits".automatika_aktivna AND "rolo_vrata_otvorena" AND NOT "Errors".error_bit);
   "Op3_zavareni_start" := ("HMI_signals".set_zavareni AND "HMI_signals".setup_mode) OR ("Sekvence_DB".Op3_zavareni_start AND "pom_bits".automatika_aktivna AND "rolo_vrata_otvorena" AND NOT "Errors".error_bit);
   "Okvir_manji_unisti_start" := ("HMI_signals".set_zavareni AND "HMI_signals".setup_mode) OR ("Sekvence_DB".Op3_zavareni_start AND "pom_bits".automatika_aktivna AND "rolo_vrata_otvorena" AND NOT "Errors".error_bit);
   "Okvir_veci_unisti_start" := ("HMI_signals".set_zavareni AND "HMI_signals".setup_mode) OR ("Sekvence_DB".Op3_zavareni_start AND "pom_bits".automatika_aktivna AND "rolo_vrata_otvorena" AND NOT "Errors".error_bit);
   "Zavareno_unisti_start" := ("Sekvence_DB".Zavareno_unisti_start AND "pom_bits".automatika_aktivna AND NOT "Errors".error_bit) OR ("HMI_signals".set_unisti_zavarene AND "HMI_signals".setup_mode);
END_REGION

REGION Network 16: Material flow 2
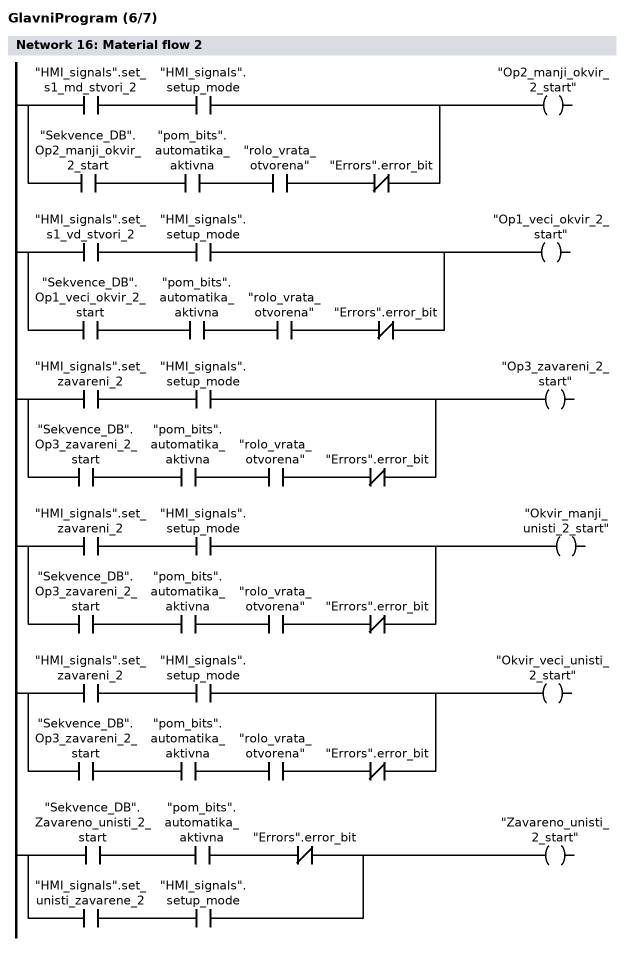
   RUNG wire#powerrail
      Contact( "HMI_signals".set_s1_md_stvori_2 )
      Contact( "HMI_signals".setup_mode )
      wire#w1
      Coil( "Op2_manji_okvir_2_start" )
   END_RUNG
   RUNG wire#powerrail
      Contact( "Sekvence_DB".Op2_manji_okvir_2_start )
      Contact( "pom_bits".automatika_aktivna )
      Contact( "rolo_vrata_otvorena" )
      I_Contact( "Errors".error_bit )
   END_RUNG wire#w1
   RUNG wire#powerrail
      Contact( "HMI_signals".set_s1_vd_stvori_2 )
      Contact( "HMI_signals".setup_mode )
      wire#w2
      Coil( "Op1_veci_okvir_2_start" )
   END_RUNG
   RUNG wire#powerrail
      Contact( "Sekvence_DB".Op1_veci_okvir_2_start )
      Contact( "pom_bits".automatika_aktivna )
      Contact( "rolo_vrata_otvorena" )
      I_Contact( "Errors".error_bit )
   END_RUNG wire#w2
   RUNG wire#powerrail
      Contact( "HMI_signals".set_zavareni_2 )
      Contact( "HMI_signals".setup_mode )
      wire#w3
      Coil( "Op3_zavareni_2_start" )
   END_RUNG
   RUNG wire#powerrail
      Contact( "Sekvence_DB".Op3_zavareni_2_start )
      Contact( "pom_bits".automatika_aktivna )
      Contact( "rolo_vrata_otvorena" )
      I_Contact( "Errors".error_bit )
   END_RUNG wire#w3
   RUNG wire#powerrail
      Contact( "HMI_signals".set_zavareni_2 )
      Contact( "HMI_signals".setup_mode )
      wire#w4
      Coil( "Okvir_manji_unisti_2_start" )
   END_RUNG
   RUNG wire#powerrail
      Contact( "Sekvence_DB".Op3_zavareni_2_start )
      Contact( "pom_bits".automatika_aktivna )
      Contact( "rolo_vrata_otvorena" )
      I_Contact( "Errors".error_bit )
   END_RUNG wire#w4
   RUNG wire#powerrail
      Contact( "HMI_signals".set_zavareni_2 )
      Contact( "HMI_signals".setup_mode )
      wire#w5
      Coil( "Okvir_veci_unisti_2_start" )
   END_RUNG
   RUNG wire#powerrail
      Contact( "Sekvence_DB".Op3_zavareni_2_start )
      Contact( "pom_bits".automatika_aktivna )
      Contact( "rolo_vrata_otvorena" )
      I_Contact( "Errors".error_bit )
   END_RUNG wire#w5
   RUNG wire#powerrail
      Contact( "Sekvence_DB".Zavareno_unisti_2_start )
      Contact( "pom_bits".automatika_aktivna )
      I_Contact( "Errors".error_bit )
      wire#w6
      Coil( "Zavareno_unisti_2_start" )
   END_RUNG
   RUNG wire#powerrail
      Contact( "HMI_signals".set_unisti_zavarene_2 )
      Contact( "HMI_signals".setup_mode )
   END_RUNG wire#w6
   // the same network as SCL:
   "Op2_manji_okvir_2_start" := ("HMI_signals".set_s1_md_stvori_2 AND "HMI_signals".setup_mode) OR ("Sekvence_DB".Op2_manji_okvir_2_start AND "pom_bits".automatika_aktivna AND "rolo_vrata_otvorena" AND NOT "Errors".error_bit);
   "Op1_veci_okvir_2_start" := ("HMI_signals".set_s1_vd_stvori_2 AND "HMI_signals".setup_mode) OR ("Sekvence_DB".Op1_veci_okvir_2_start AND "pom_bits".automatika_aktivna AND "rolo_vrata_otvorena" AND NOT "Errors".error_bit);
   "Op3_zavareni_2_start" := ("HMI_signals".set_zavareni_2 AND "HMI_signals".setup_mode) OR ("Sekvence_DB".Op3_zavareni_2_start AND "pom_bits".automatika_aktivna AND "rolo_vrata_otvorena" AND NOT "Errors".error_bit);
   "Okvir_manji_unisti_2_start" := ("HMI_signals".set_zavareni_2 AND "HMI_signals".setup_mode) OR ("Sekvence_DB".Op3_zavareni_2_start AND "pom_bits".automatika_aktivna AND "rolo_vrata_otvorena" AND NOT "Errors".error_bit);
   "Okvir_veci_unisti_2_start" := ("HMI_signals".set_zavareni_2 AND "HMI_signals".setup_mode) OR ("Sekvence_DB".Op3_zavareni_2_start AND "pom_bits".automatika_aktivna AND "rolo_vrata_otvorena" AND NOT "Errors".error_bit);
   "Zavareno_unisti_2_start" := ("Sekvence_DB".Zavareno_unisti_2_start AND "pom_bits".automatika_aktivna AND NOT "Errors".error_bit) OR ("HMI_signals".set_unisti_zavarene_2 AND "HMI_signals".setup_mode);
END_REGION

REGION Network 17: Semafor
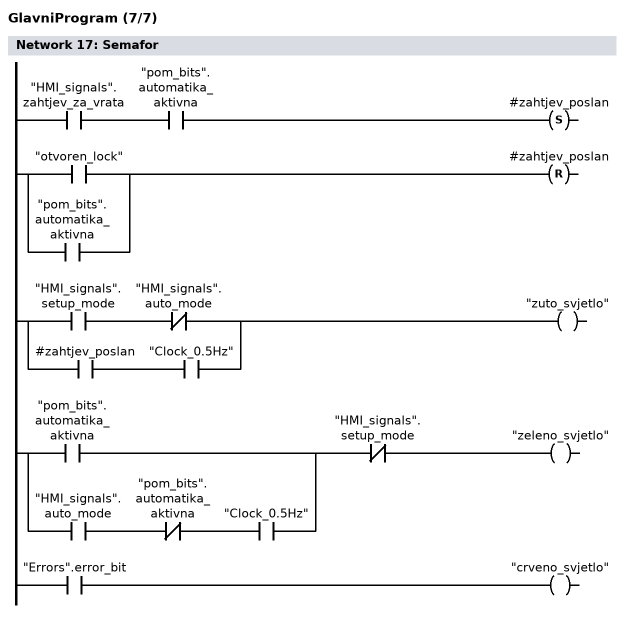
   RUNG wire#powerrail
      Contact( "HMI_signals".zahtjev_za_vrata )
      Contact( "pom_bits".automatika_aktivna )
      S_Coil( #zahtjev_poslan )
   END_RUNG
   RUNG wire#powerrail
      Contact( "otvoren_lock" )
      wire#w1
      R_Coil( #zahtjev_poslan )
   END_RUNG
   RUNG wire#powerrail
      Contact( "pom_bits".automatika_aktivna )
   END_RUNG wire#w1
   RUNG wire#powerrail
      Contact( "HMI_signals".setup_mode )
      I_Contact( "HMI_signals".auto_mode )
      wire#w2
      Coil( "zuto_svjetlo" )
   END_RUNG
   RUNG wire#powerrail
      Contact( #zahtjev_poslan )
      Contact( "Clock_0.5Hz" )
   END_RUNG wire#w2
   RUNG wire#powerrail
      Contact( "pom_bits".automatika_aktivna )
      wire#w3
      I_Contact( "HMI_signals".setup_mode )
      Coil( "zeleno_svjetlo" )
   END_RUNG
   RUNG wire#powerrail
      Contact( "HMI_signals".auto_mode )
      I_Contact( "pom_bits".automatika_aktivna )
      Contact( "Clock_0.5Hz" )
   END_RUNG wire#w3
   RUNG wire#powerrail
      Contact( "Errors".error_bit )
      Coil( "crveno_svjetlo" )
   END_RUNG
   // the same network as SCL:
   IF "HMI_signals".zahtjev_za_vrata AND "pom_bits".automatika_aktivna THEN #zahtjev_poslan := TRUE; END_IF;
   IF "otvoren_lock" OR "pom_bits".automatika_aktivna THEN #zahtjev_poslan := FALSE; END_IF;
   "zuto_svjetlo" := ("HMI_signals".setup_mode AND NOT "HMI_signals".auto_mode) OR (#zahtjev_poslan AND "Clock_0.5Hz");
   "zeleno_svjetlo" := ("pom_bits".automatika_aktivna OR ("HMI_signals".auto_mode AND NOT "pom_bits".automatika_aktivna AND "Clock_0.5Hz")) AND NOT "HMI_signals".setup_mode;
   "crveno_svjetlo" := "Errors".error_bit;
END_REGION
END_FUNCTION_BLOCK

// folder: Sekvence

FUNCTION_BLOCK "Okretni_stol_sekvenca"   // FB3, LAD
{ S7_Optimized_Access := 'TRUE' }
VERSION : 0.1
   VAR_INPUT
      inicijalizacija : Bool;
   END_VAR
   VAR
      stepNum : Int;
      stepNumPrev : Int;
      bit_na_brid : Array[0..2] of Bool;
   END_VAR
   VAR_TEMP
      "nop" : Bool;
   END_VAR
   VAR_TEMP   // added for the SCL form of the ladder/FBD networks
      _w1 : Bool;
   END_VAR
BEGIN

REGION Network 1: Inicijalizacija sekvence
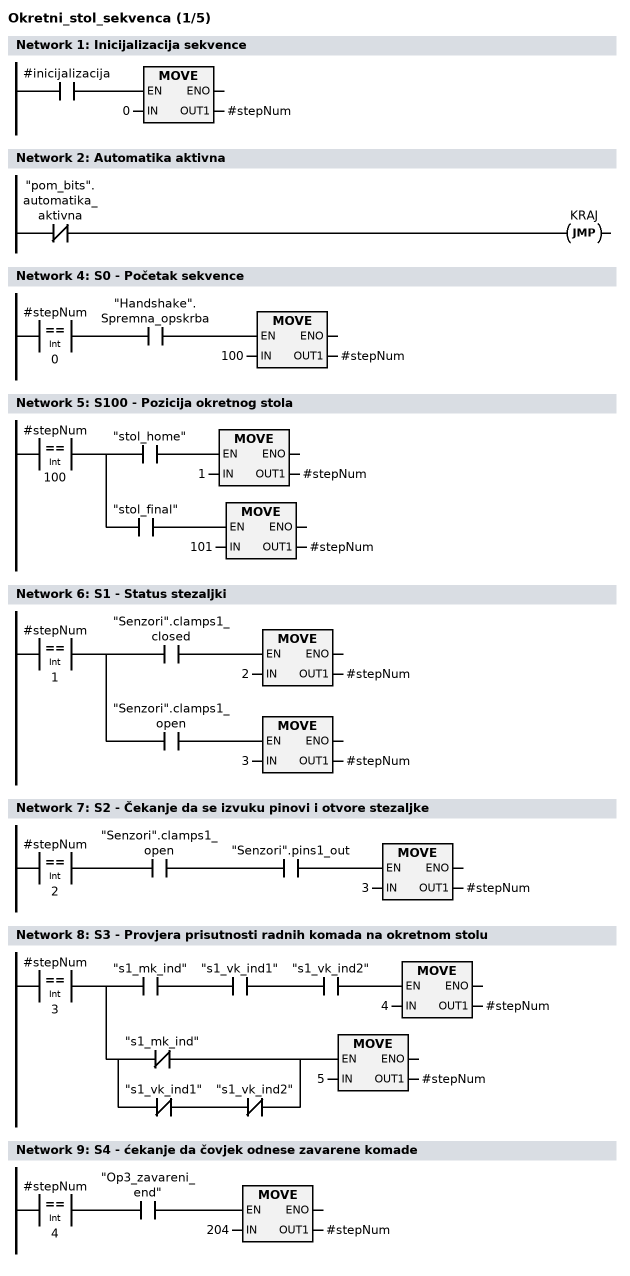
   RUNG wire#powerrail
      Contact( #inicijalizacija )
      Move(in := 0, out1 => #stepNum)
   END_RUNG
   // the same network as SCL:
   IF #inicijalizacija THEN #stepNum := 0; END_IF;
END_REGION

REGION Network 2: Automatika aktivna
   RUNG wire#powerrail
      I_Contact( "pom_bits".automatika_aktivna )
      JumpCoil( KRAJ )
   END_RUNG
   // the same network as SCL:
   IF NOT "pom_bits".automatika_aktivna THEN GOTO KRAJ; END_IF;
END_REGION

REGION Network 3: KORACI: 1 - stol u početnoj poziciji, 101 - stol u okrenutoj poziciji
END_REGION

REGION Network 4: S0 - Početak sekvence
   RUNG wire#powerrail
      { S7_Templates := "SrcType := Int" } EQ_Contact(in1 := #stepNum, in2 := 0)
      Contact( "Handshake".Spremna_opskrba )
      Move(in := 100, out1 => #stepNum)
   END_RUNG
   // the same network as SCL:
   IF (#stepNum = 0) AND "Handshake".Spremna_opskrba THEN #stepNum := 100; END_IF;
END_REGION

REGION Network 5: S100 - Pozicija okretnog stola
   RUNG wire#powerrail
      { S7_Templates := "SrcType := Int" } EQ_Contact(in1 := #stepNum, in2 := 100)
      wire#w1
      Contact( "stol_home" )
      Move(in := 1, out1 => #stepNum)
   END_RUNG
   RUNG wire#w1
      Contact( "stol_final" )
      Move(in := 101, out1 => #stepNum)
   END_RUNG
   // the same network as SCL:
   #_w1 := #stepNum = 100;
   IF #_w1 AND "stol_home" THEN #stepNum := 1; END_IF;
   IF #_w1 AND "stol_final" THEN #stepNum := 101; END_IF;
END_REGION

REGION Network 6: S1 - Status stezaljki
   RUNG wire#powerrail
      { S7_Templates := "SrcType := Int" } EQ_Contact(in1 := #stepNum, in2 := 1)
      wire#w1
      Contact( "Senzori".clamps1_closed )
      Move(in := 2, out1 => #stepNum)
   END_RUNG
   RUNG wire#w1
      Contact( "Senzori".clamps1_open )
      Move(in := 3, out1 => #stepNum)
   END_RUNG
   // the same network as SCL:
   #_w1 := #stepNum = 1;
   IF #_w1 AND "Senzori".clamps1_closed THEN #stepNum := 2; END_IF;
   IF #_w1 AND "Senzori".clamps1_open THEN #stepNum := 3; END_IF;
END_REGION

REGION Network 7: S2 - Čekanje da se izvuku pinovi i otvore stezaljke
   RUNG wire#powerrail
      { S7_Templates := "SrcType := Int" } EQ_Contact(in1 := #stepNum, in2 := 2)
      Contact( "Senzori".clamps1_open )
      Contact( "Senzori".pins1_out )
      Move(in := 3, out1 => #stepNum)
   END_RUNG
   // the same network as SCL:
   IF (#stepNum = 2) AND "Senzori".clamps1_open AND "Senzori".pins1_out THEN #stepNum := 3; END_IF;
END_REGION

REGION Network 8: S3 - Provjera prisutnosti radnih komada na okretnom stolu
   RUNG wire#powerrail
      { S7_Templates := "SrcType := Int" } EQ_Contact(in1 := #stepNum, in2 := 3)
      wire#w1
      Contact( "s1_mk_ind" )
      Contact( "s1_vk_ind1" )
      Contact( "s1_vk_ind2" )
      Move(in := 4, out1 => #stepNum)
   END_RUNG
   RUNG wire#w1
      I_Contact( "s1_mk_ind" )
      wire#w2
      Move(in := 5, out1 => #stepNum)
   END_RUNG
   RUNG wire#w1
      I_Contact( "s1_vk_ind1" )
      I_Contact( "s1_vk_ind2" )
   END_RUNG wire#w2
   // the same network as SCL:
   #_w1 := #stepNum = 3;
   IF #_w1 AND "s1_mk_ind" AND "s1_vk_ind1" AND "s1_vk_ind2" THEN #stepNum := 4; END_IF;
   IF #_w1 AND (NOT "s1_mk_ind" OR (NOT "s1_vk_ind1" AND NOT "s1_vk_ind2")) THEN #stepNum := 5; END_IF;
END_REGION

REGION Network 9: S4 - ćekanje da čovjek odnese zavarene komade
   RUNG wire#powerrail
      { S7_Templates := "SrcType := Int" } EQ_Contact(in1 := #stepNum, in2 := 4)
      Contact( "Op3_zavareni_end" )
      Move(in := 204, out1 => #stepNum)
   END_RUNG
   // the same network as SCL:
   IF (#stepNum = 4) AND "Op3_zavareni_end" THEN #stepNum := 204; END_IF;
END_REGION

REGION Network 10: S204 - Uklanjanje zavarenih predmeta
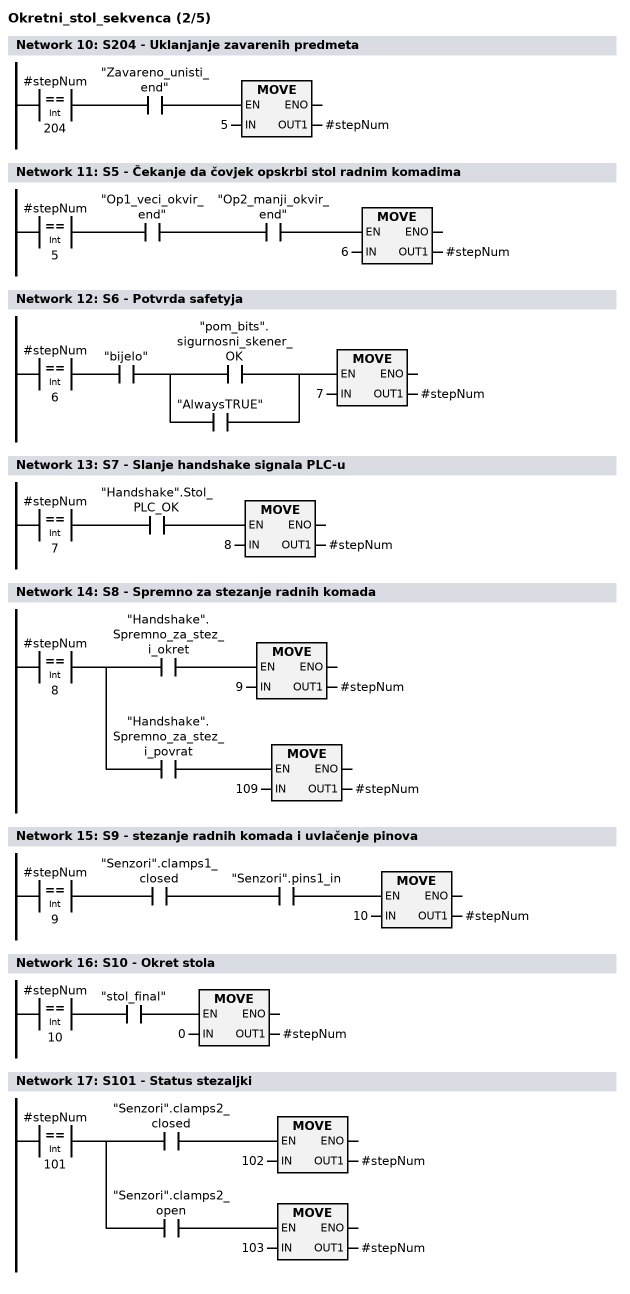
   RUNG wire#powerrail
      { S7_Templates := "SrcType := Int" } EQ_Contact(in1 := #stepNum, in2 := 204)
      Contact( "Zavareno_unisti_end" )
      Move(in := 5, out1 => #stepNum)
   END_RUNG
   // the same network as SCL:
   IF (#stepNum = 204) AND "Zavareno_unisti_end" THEN #stepNum := 5; END_IF;
END_REGION

REGION Network 11: S5 - Čekanje da čovjek opskrbi stol radnim komadima
   RUNG wire#powerrail
      { S7_Templates := "SrcType := Int" } EQ_Contact(in1 := #stepNum, in2 := 5)
      Contact( "Op1_veci_okvir_end" )
      Contact( "Op2_manji_okvir_end" )
      Move(in := 6, out1 => #stepNum)
   END_RUNG
   // the same network as SCL:
   IF (#stepNum = 5) AND "Op1_veci_okvir_end" AND "Op2_manji_okvir_end" THEN #stepNum := 6; END_IF;
END_REGION

REGION Network 12: S6 - Potvrda safetyja
   RUNG wire#powerrail
      { S7_Templates := "SrcType := Int" } EQ_Contact(in1 := #stepNum, in2 := 6)
      Contact( "bijelo" )
      wire#w1
      Contact( "pom_bits".sigurnosni_skener_OK )
      wire#w2
      Move(in := 7, out1 => #stepNum)
   END_RUNG
   RUNG wire#w1
      Contact( "AlwaysTRUE" )
   END_RUNG wire#w2
   // the same network as SCL:
   IF (#stepNum = 6) AND "bijelo" AND ("pom_bits".sigurnosni_skener_OK OR "AlwaysTRUE") THEN
       #stepNum := 7;
   END_IF;
END_REGION

REGION Network 13: S7 - Slanje handshake signala PLC-u
   RUNG wire#powerrail
      { S7_Templates := "SrcType := Int" } EQ_Contact(in1 := #stepNum, in2 := 7)
      Contact( "Handshake".Stol_PLC_OK )
      Move(in := 8, out1 => #stepNum)
   END_RUNG
   // the same network as SCL:
   IF (#stepNum = 7) AND "Handshake".Stol_PLC_OK THEN #stepNum := 8; END_IF;
END_REGION

REGION Network 14: S8 - Spremno za stezanje radnih komada
   RUNG wire#powerrail
      { S7_Templates := "SrcType := Int" } EQ_Contact(in1 := #stepNum, in2 := 8)
      wire#w1
      Contact( "Handshake".Spremno_za_stez_i_okret )
      Move(in := 9, out1 => #stepNum)
   END_RUNG
   RUNG wire#w1
      Contact( "Handshake".Spremno_za_stez_i_povrat )
      Move(in := 109, out1 => #stepNum)
   END_RUNG
   // the same network as SCL:
   #_w1 := #stepNum = 8;
   IF #_w1 AND "Handshake".Spremno_za_stez_i_okret THEN #stepNum := 9; END_IF;
   IF #_w1 AND "Handshake".Spremno_za_stez_i_povrat THEN #stepNum := 109; END_IF;
END_REGION

REGION Network 15: S9 - stezanje radnih komada i uvlačenje pinova
   RUNG wire#powerrail
      { S7_Templates := "SrcType := Int" } EQ_Contact(in1 := #stepNum, in2 := 9)
      Contact( "Senzori".clamps1_closed )
      Contact( "Senzori".pins1_in )
      Move(in := 10, out1 => #stepNum)
   END_RUNG
   // the same network as SCL:
   IF (#stepNum = 9) AND "Senzori".clamps1_closed AND "Senzori".pins1_in THEN #stepNum := 10; END_IF;
END_REGION

REGION Network 16: S10 - Okret stola
   RUNG wire#powerrail
      { S7_Templates := "SrcType := Int" } EQ_Contact(in1 := #stepNum, in2 := 10)
      Contact( "stol_final" )
      Move(in := 0, out1 => #stepNum)
   END_RUNG
   // the same network as SCL:
   IF (#stepNum = 10) AND "stol_final" THEN #stepNum := 0; END_IF;
END_REGION

REGION Network 17: S101 - Status stezaljki
   RUNG wire#powerrail
      { S7_Templates := "SrcType := Int" } EQ_Contact(in1 := #stepNum, in2 := 101)
      wire#w1
      Contact( "Senzori".clamps2_closed )
      Move(in := 102, out1 => #stepNum)
   END_RUNG
   RUNG wire#w1
      Contact( "Senzori".clamps2_open )
      Move(in := 103, out1 => #stepNum)
   END_RUNG
   // the same network as SCL:
   #_w1 := #stepNum = 101;
   IF #_w1 AND "Senzori".clamps2_closed THEN #stepNum := 102; END_IF;
   IF #_w1 AND "Senzori".clamps2_open THEN #stepNum := 103; END_IF;
END_REGION

REGION Network 18: S102 - Čekanje da se pinovi izvuku i otvore stezaljke
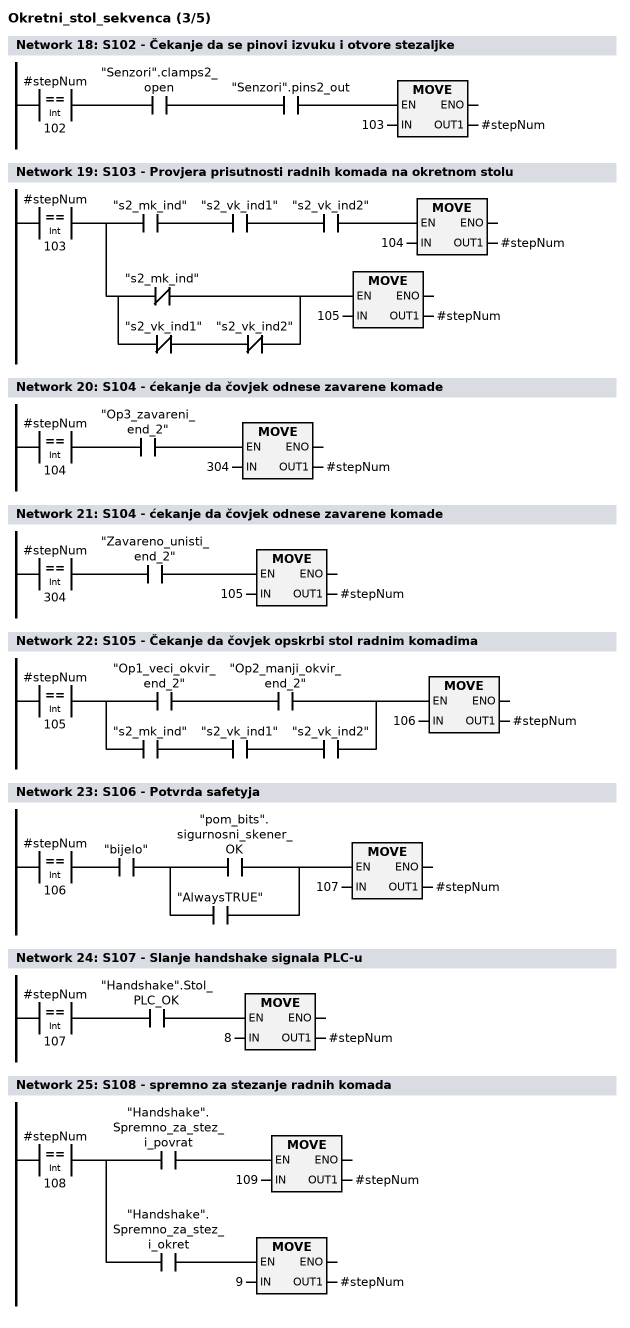
   RUNG wire#powerrail
      { S7_Templates := "SrcType := Int" } EQ_Contact(in1 := #stepNum, in2 := 102)
      Contact( "Senzori".clamps2_open )
      Contact( "Senzori".pins2_out )
      Move(in := 103, out1 => #stepNum)
   END_RUNG
   // the same network as SCL:
   IF (#stepNum = 102) AND "Senzori".clamps2_open AND "Senzori".pins2_out THEN #stepNum := 103; END_IF;
END_REGION

REGION Network 19: S103 - Provjera prisutnosti radnih komada na okretnom stolu
   RUNG wire#powerrail
      { S7_Templates := "SrcType := Int" } EQ_Contact(in1 := #stepNum, in2 := 103)
      wire#w1
      Contact( "s2_mk_ind" )
      Contact( "s2_vk_ind1" )
      Contact( "s2_vk_ind2" )
      Move(in := 104, out1 => #stepNum)
   END_RUNG
   RUNG wire#w1
      I_Contact( "s2_mk_ind" )
      wire#w2
      Move(in := 105, out1 => #stepNum)
   END_RUNG
   RUNG wire#w1
      I_Contact( "s2_vk_ind1" )
      I_Contact( "s2_vk_ind2" )
   END_RUNG wire#w2
   // the same network as SCL:
   #_w1 := #stepNum = 103;
   IF #_w1 AND "s2_mk_ind" AND "s2_vk_ind1" AND "s2_vk_ind2" THEN #stepNum := 104; END_IF;
   IF #_w1 AND (NOT "s2_mk_ind" OR (NOT "s2_vk_ind1" AND NOT "s2_vk_ind2")) THEN #stepNum := 105; END_IF;
END_REGION

REGION Network 20: S104 - ćekanje da čovjek odnese zavarene komade
   RUNG wire#powerrail
      { S7_Templates := "SrcType := Int" } EQ_Contact(in1 := #stepNum, in2 := 104)
      Contact( "Op3_zavareni_end_2" )
      Move(in := 304, out1 => #stepNum)
   END_RUNG
   // the same network as SCL:
   IF (#stepNum = 104) AND "Op3_zavareni_end_2" THEN #stepNum := 304; END_IF;
END_REGION

REGION Network 21: S104 - ćekanje da čovjek odnese zavarene komade
   RUNG wire#powerrail
      { S7_Templates := "SrcType := Int" } EQ_Contact(in1 := #stepNum, in2 := 304)
      Contact( "Zavareno_unisti_end_2" )
      Move(in := 105, out1 => #stepNum)
   END_RUNG
   // the same network as SCL:
   IF (#stepNum = 304) AND "Zavareno_unisti_end_2" THEN #stepNum := 105; END_IF;
END_REGION

REGION Network 22: S105 - Čekanje da čovjek opskrbi stol radnim komadima
   RUNG wire#powerrail
      { S7_Templates := "SrcType := Int" } EQ_Contact(in1 := #stepNum, in2 := 105)
      wire#w1
      Contact( "Op1_veci_okvir_end_2" )
      Contact( "Op2_manji_okvir_end_2" )
      wire#w2
      Move(in := 106, out1 => #stepNum)
   END_RUNG
   RUNG wire#w1
      Contact( "s2_mk_ind" )
      Contact( "s2_vk_ind1" )
      Contact( "s2_vk_ind2" )
   END_RUNG wire#w2
   // the same network as SCL:
   IF (#stepNum = 105) AND (("Op1_veci_okvir_end_2" AND "Op2_manji_okvir_end_2") OR ("s2_mk_ind" AND "s2_vk_ind1" AND "s2_vk_ind2")) THEN
       #stepNum := 106;
   END_IF;
END_REGION

REGION Network 23: S106 - Potvrda safetyja
   RUNG wire#powerrail
      { S7_Templates := "SrcType := Int" } EQ_Contact(in1 := #stepNum, in2 := 106)
      Contact( "bijelo" )
      wire#w1
      Contact( "pom_bits".sigurnosni_skener_OK )
      wire#w2
      Move(in := 107, out1 => #stepNum)
   END_RUNG
   RUNG wire#w1
      Contact( "AlwaysTRUE" )
   END_RUNG wire#w2
   // the same network as SCL:
   IF (#stepNum = 106) AND "bijelo" AND ("pom_bits".sigurnosni_skener_OK OR "AlwaysTRUE") THEN
       #stepNum := 107;
   END_IF;
END_REGION

REGION Network 24: S107 - Slanje handshake signala PLC-u
   RUNG wire#powerrail
      { S7_Templates := "SrcType := Int" } EQ_Contact(in1 := #stepNum, in2 := 107)
      Contact( "Handshake".Stol_PLC_OK )
      Move(in := 8, out1 => #stepNum)
   END_RUNG
   // the same network as SCL:
   IF (#stepNum = 107) AND "Handshake".Stol_PLC_OK THEN #stepNum := 8; END_IF;
END_REGION

REGION Network 25: S108 - spremno za stezanje radnih komada
   RUNG wire#powerrail
      { S7_Templates := "SrcType := Int" } EQ_Contact(in1 := #stepNum, in2 := 108)
      wire#w1
      Contact( "Handshake".Spremno_za_stez_i_povrat )
      Move(in := 109, out1 => #stepNum)
   END_RUNG
   RUNG wire#w1
      Contact( "Handshake".Spremno_za_stez_i_okret )
      Move(in := 9, out1 => #stepNum)
   END_RUNG
   // the same network as SCL:
   #_w1 := #stepNum = 108;
   IF #_w1 AND "Handshake".Spremno_za_stez_i_povrat THEN #stepNum := 109; END_IF;
   IF #_w1 AND "Handshake".Spremno_za_stez_i_okret THEN #stepNum := 9; END_IF;
END_REGION

REGION Network 26: S109 - stezanje radnih komada i uvlačenje pinova
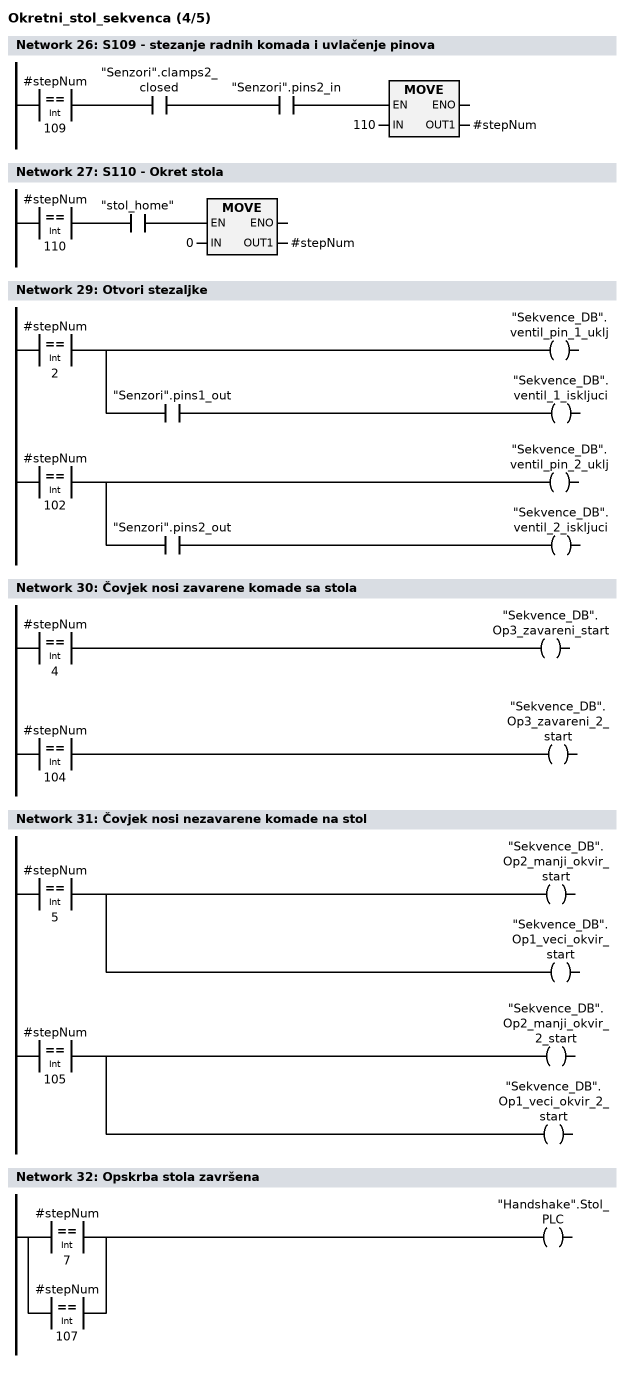
   RUNG wire#powerrail
      { S7_Templates := "SrcType := Int" } EQ_Contact(in1 := #stepNum, in2 := 109)
      Contact( "Senzori".clamps2_closed )
      Contact( "Senzori".pins2_in )
      Move(in := 110, out1 => #stepNum)
   END_RUNG
   // the same network as SCL:
   IF (#stepNum = 109) AND "Senzori".clamps2_closed AND "Senzori".pins2_in THEN #stepNum := 110; END_IF;
END_REGION

REGION Network 27: S110 - Okret stola
   RUNG wire#powerrail
      { S7_Templates := "SrcType := Int" } EQ_Contact(in1 := #stepNum, in2 := 110)
      Contact( "stol_home" )
      Move(in := 0, out1 => #stepNum)
   END_RUNG
   // the same network as SCL:
   IF (#stepNum = 110) AND "stol_home" THEN #stepNum := 0; END_IF;
END_REGION

REGION Network 28: RADNJE
END_REGION

REGION Network 29: Otvori stezaljke
   RUNG wire#powerrail
      { S7_Templates := "SrcType := Int" } EQ_Contact(in1 := #stepNum, in2 := 2)
      wire#w1
      Coil( "Sekvence_DB".ventil_pin_1_uklj )
   END_RUNG
   RUNG wire#w1
      Contact( "Senzori".pins1_out )
      Coil( "Sekvence_DB".ventil_1_iskljuci )
   END_RUNG
   RUNG wire#powerrail
      { S7_Templates := "SrcType := Int" } EQ_Contact(in1 := #stepNum, in2 := 102)
      wire#w2
      Coil( "Sekvence_DB".ventil_pin_2_uklj )
   END_RUNG
   RUNG wire#w2
      Contact( "Senzori".pins2_out )
      Coil( "Sekvence_DB".ventil_2_iskljuci )
   END_RUNG
   // the same network as SCL:
   "Sekvence_DB".ventil_pin_1_uklj := #stepNum = 2;
   "Sekvence_DB".ventil_1_iskljuci := "Sekvence_DB".ventil_pin_1_uklj AND "Senzori".pins1_out;
   "Sekvence_DB".ventil_pin_2_uklj := #stepNum = 102;
   "Sekvence_DB".ventil_2_iskljuci := "Sekvence_DB".ventil_pin_2_uklj AND "Senzori".pins2_out;
END_REGION

REGION Network 30: Čovjek nosi zavarene komade sa stola
   RUNG wire#powerrail
      { S7_Templates := "SrcType := Int" } EQ_Contact(in1 := #stepNum, in2 := 4)
      Coil( "Sekvence_DB".Op3_zavareni_start )
   END_RUNG
   RUNG wire#powerrail
      { S7_Templates := "SrcType := Int" } EQ_Contact(in1 := #stepNum, in2 := 104)
      Coil( "Sekvence_DB".Op3_zavareni_2_start )
   END_RUNG
   // the same network as SCL:
   "Sekvence_DB".Op3_zavareni_start := #stepNum = 4;
   "Sekvence_DB".Op3_zavareni_2_start := #stepNum = 104;
END_REGION

REGION Network 31: Čovjek nosi nezavarene komade na stol
   RUNG wire#powerrail
      { S7_Templates := "SrcType := Int" } EQ_Contact(in1 := #stepNum, in2 := 5)
      wire#w1
      Coil( "Sekvence_DB".Op2_manji_okvir_start )
   END_RUNG
   RUNG wire#w1
      Coil( "Sekvence_DB".Op1_veci_okvir_start )
   END_RUNG
   RUNG wire#powerrail
      { S7_Templates := "SrcType := Int" } EQ_Contact(in1 := #stepNum, in2 := 105)
      wire#w2
      Coil( "Sekvence_DB".Op2_manji_okvir_2_start )
   END_RUNG
   RUNG wire#w2
      Coil( "Sekvence_DB".Op1_veci_okvir_2_start )
   END_RUNG
   // the same network as SCL:
   "Sekvence_DB".Op2_manji_okvir_start := #stepNum = 5;
   "Sekvence_DB".Op1_veci_okvir_start := "Sekvence_DB".Op2_manji_okvir_start;
   "Sekvence_DB".Op2_manji_okvir_2_start := #stepNum = 105;
   "Sekvence_DB".Op1_veci_okvir_2_start := "Sekvence_DB".Op2_manji_okvir_2_start;
END_REGION

REGION Network 32: Opskrba stola završena
   RUNG wire#powerrail
      { S7_Templates := "SrcType := Int" } EQ_Contact(in1 := #stepNum, in2 := 7)
      wire#w1
      Coil( "Handshake".Stol_PLC )
   END_RUNG
   RUNG wire#powerrail
      { S7_Templates := "SrcType := Int" } EQ_Contact(in1 := #stepNum, in2 := 107)
   END_RUNG wire#w1
   // the same network as SCL:
   "Handshake".Stol_PLC := (#stepNum = 7) OR (#stepNum = 107);
END_REGION

REGION Network 33: Stezanje radnih komada
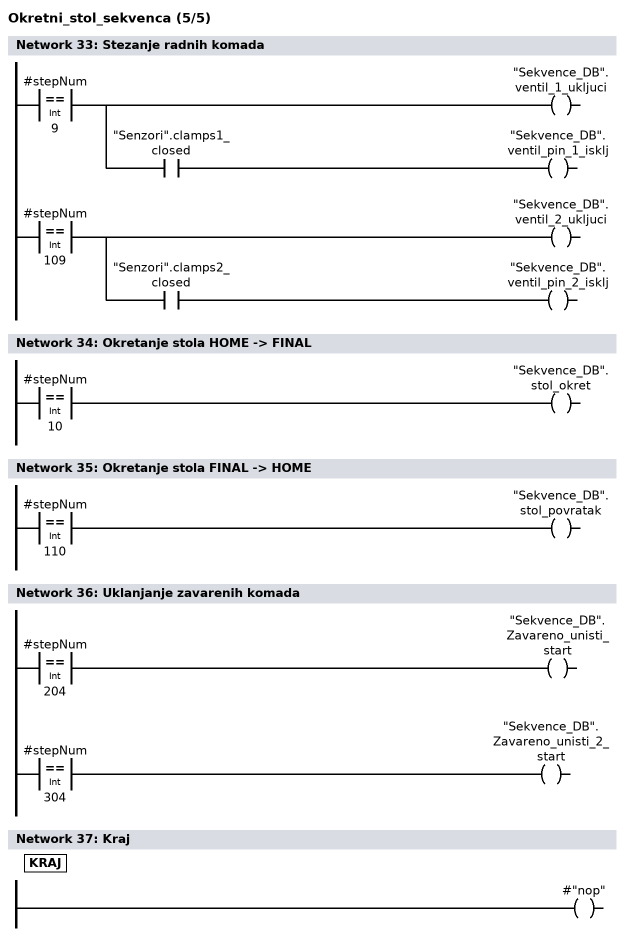
   RUNG wire#powerrail
      { S7_Templates := "SrcType := Int" } EQ_Contact(in1 := #stepNum, in2 := 9)
      wire#w1
      Coil( "Sekvence_DB".ventil_1_ukljuci )
   END_RUNG
   RUNG wire#w1
      Contact( "Senzori".clamps1_closed )
      Coil( "Sekvence_DB".ventil_pin_1_isklj )
   END_RUNG
   RUNG wire#powerrail
      { S7_Templates := "SrcType := Int" } EQ_Contact(in1 := #stepNum, in2 := 109)
      wire#w2
      Coil( "Sekvence_DB".ventil_2_ukljuci )
   END_RUNG
   RUNG wire#w2
      Contact( "Senzori".clamps2_closed )
      Coil( "Sekvence_DB".ventil_pin_2_isklj )
   END_RUNG
   // the same network as SCL:
   "Sekvence_DB".ventil_1_ukljuci := #stepNum = 9;
   "Sekvence_DB".ventil_pin_1_isklj := "Sekvence_DB".ventil_1_ukljuci AND "Senzori".clamps1_closed;
   "Sekvence_DB".ventil_2_ukljuci := #stepNum = 109;
   "Sekvence_DB".ventil_pin_2_isklj := "Sekvence_DB".ventil_2_ukljuci AND "Senzori".clamps2_closed;
END_REGION

REGION Network 34: Okretanje stola HOME -> FINAL
   RUNG wire#powerrail
      { S7_Templates := "SrcType := Int" } EQ_Contact(in1 := #stepNum, in2 := 10)
      Coil( "Sekvence_DB".stol_okret )
   END_RUNG
   // the same network as SCL:
   "Sekvence_DB".stol_okret := #stepNum = 10;
END_REGION

REGION Network 35: Okretanje stola FINAL -> HOME
   RUNG wire#powerrail
      { S7_Templates := "SrcType := Int" } EQ_Contact(in1 := #stepNum, in2 := 110)
      Coil( "Sekvence_DB".stol_povratak )
   END_RUNG
   // the same network as SCL:
   "Sekvence_DB".stol_povratak := #stepNum = 110;
END_REGION

REGION Network 36: Uklanjanje zavarenih komada
   RUNG wire#powerrail
      { S7_Templates := "SrcType := Int" } EQ_Contact(in1 := #stepNum, in2 := 204)
      Coil( "Sekvence_DB".Zavareno_unisti_start )
   END_RUNG
   RUNG wire#powerrail
      { S7_Templates := "SrcType := Int" } EQ_Contact(in1 := #stepNum, in2 := 304)
      Coil( "Sekvence_DB".Zavareno_unisti_2_start )
   END_RUNG
   // the same network as SCL:
   "Sekvence_DB".Zavareno_unisti_start := #stepNum = 204;
   "Sekvence_DB".Zavareno_unisti_2_start := #stepNum = 304;
END_REGION

REGION Network 37: Kraj
   Label( KRAJ )
   RUNG wire#powerrail
      Coil( #"nop" )
   END_RUNG
   // the same network as SCL:
   KRAJ:
   #"nop" := TRUE;
END_REGION
END_FUNCTION_BLOCK

FUNCTION_BLOCK "Glavna_sekvenca"   // FB4, LAD
{ S7_Optimized_Access := 'TRUE' }
VERSION : 0.1
   VAR_INPUT
      inicijalizacija : Bool;
   END_VAR
   VAR
      stepNum : Int;
      bit_na_brid : Array[0..4] of Bool;
      stepNumPrev : Int;
      safety_OK : Bool;
   END_VAR
   VAR_TEMP
      "nop" : Bool;
   END_VAR
   VAR_TEMP   // added for the SCL form of the ladder/FBD networks
      _w1 : Bool;
   END_VAR
BEGIN

REGION Network 1: Inicijalizacija sekvence
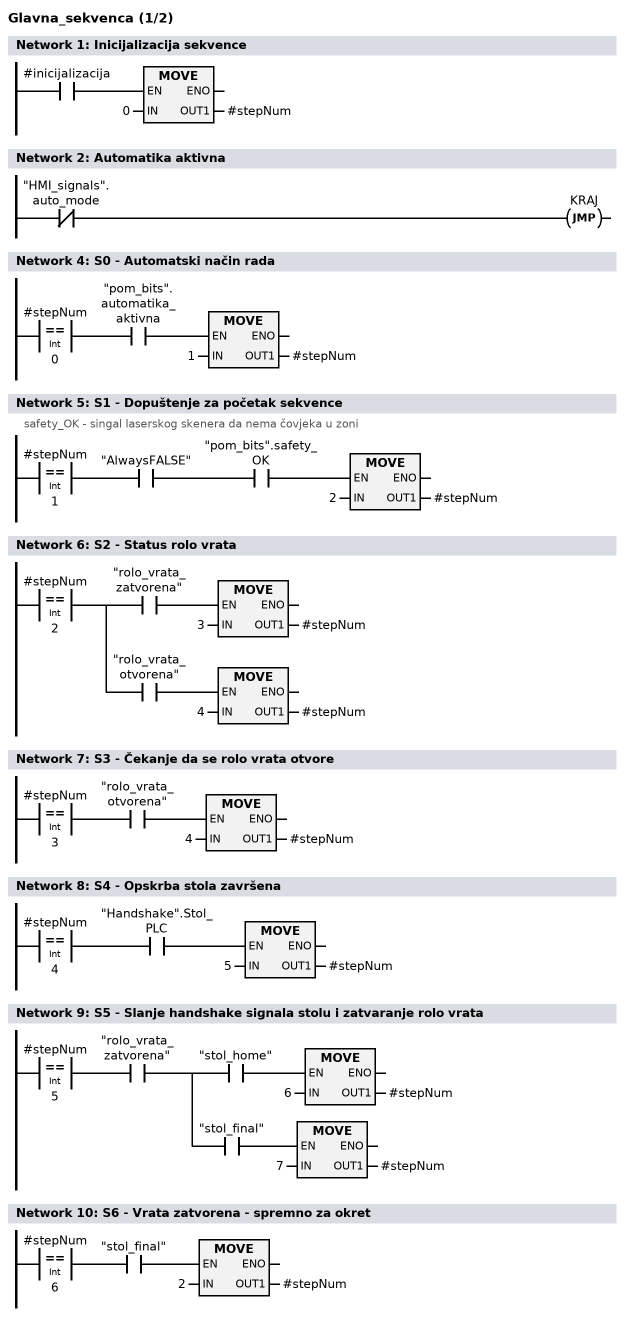
   RUNG wire#powerrail
      Contact( #inicijalizacija )
      Move(in := 0, out1 => #stepNum)
   END_RUNG
   // the same network as SCL:
   IF #inicijalizacija THEN #stepNum := 0; END_IF;
END_REGION

REGION Network 2: Automatika aktivna
   RUNG wire#powerrail
      I_Contact( "HMI_signals".auto_mode )
      JumpCoil( KRAJ )
   END_RUNG
   // the same network as SCL:
   IF NOT "HMI_signals".auto_mode THEN GOTO KRAJ; END_IF;
END_REGION

REGION Network 3: KORACI
END_REGION

REGION Network 4: S0 - Automatski način rada
   RUNG wire#powerrail
      { S7_Templates := "SrcType := Int" } EQ_Contact(in1 := #stepNum, in2 := 0)
      Contact( "pom_bits".automatika_aktivna )
      Move(in := 1, out1 => #stepNum)
   END_RUNG
   // the same network as SCL:
   IF (#stepNum = 0) AND "pom_bits".automatika_aktivna THEN #stepNum := 1; END_IF;
END_REGION

REGION Network 5: S1 - Dopuštenje za početak sekvence
   // safety_OK - singal laserskog skenera da nema čovjeka u zoni
   RUNG wire#powerrail
      { S7_Templates := "SrcType := Int" } EQ_Contact(in1 := #stepNum, in2 := 1)
      Contact( "AlwaysFALSE" )
      Contact( "pom_bits".safety_OK )
      Move(in := 2, out1 => #stepNum)
   END_RUNG
   // the same network as SCL:
   IF (#stepNum = 1) AND "AlwaysFALSE" AND "pom_bits".safety_OK THEN #stepNum := 2; END_IF;
END_REGION

REGION Network 6: S2 - Status rolo vrata
   RUNG wire#powerrail
      { S7_Templates := "SrcType := Int" } EQ_Contact(in1 := #stepNum, in2 := 2)
      wire#w1
      Contact( "rolo_vrata_zatvorena" )
      Move(in := 3, out1 => #stepNum)
   END_RUNG
   RUNG wire#w1
      Contact( "rolo_vrata_otvorena" )
      Move(in := 4, out1 => #stepNum)
   END_RUNG
   // the same network as SCL:
   #_w1 := #stepNum = 2;
   IF #_w1 AND "rolo_vrata_zatvorena" THEN #stepNum := 3; END_IF;
   IF #_w1 AND "rolo_vrata_otvorena" THEN #stepNum := 4; END_IF;
END_REGION

REGION Network 7: S3 - Čekanje da se rolo vrata otvore
   RUNG wire#powerrail
      { S7_Templates := "SrcType := Int" } EQ_Contact(in1 := #stepNum, in2 := 3)
      Contact( "rolo_vrata_otvorena" )
      Move(in := 4, out1 => #stepNum)
   END_RUNG
   // the same network as SCL:
   IF (#stepNum = 3) AND "rolo_vrata_otvorena" THEN #stepNum := 4; END_IF;
END_REGION

REGION Network 8: S4 - Opskrba stola završena
   RUNG wire#powerrail
      { S7_Templates := "SrcType := Int" } EQ_Contact(in1 := #stepNum, in2 := 4)
      Contact( "Handshake".Stol_PLC )
      Move(in := 5, out1 => #stepNum)
   END_RUNG
   // the same network as SCL:
   IF (#stepNum = 4) AND "Handshake".Stol_PLC THEN #stepNum := 5; END_IF;
END_REGION

REGION Network 9: S5 - Slanje handshake signala stolu i zatvaranje rolo vrata
   RUNG wire#powerrail
      { S7_Templates := "SrcType := Int" } EQ_Contact(in1 := #stepNum, in2 := 5)
      Contact( "rolo_vrata_zatvorena" )
      wire#w1
      Contact( "stol_home" )
      Move(in := 6, out1 => #stepNum)
   END_RUNG
   RUNG wire#w1
      Contact( "stol_final" )
      Move(in := 7, out1 => #stepNum)
   END_RUNG
   // the same network as SCL:
   #_w1 := (#stepNum = 5) AND "rolo_vrata_zatvorena";
   IF #_w1 AND "stol_home" THEN #stepNum := 6; END_IF;
   IF #_w1 AND "stol_final" THEN #stepNum := 7; END_IF;
END_REGION

REGION Network 10: S6 - Vrata zatvorena - spremno za okret
   RUNG wire#powerrail
      { S7_Templates := "SrcType := Int" } EQ_Contact(in1 := #stepNum, in2 := 6)
      Contact( "stol_final" )
      Move(in := 2, out1 => #stepNum)
   END_RUNG
   // the same network as SCL:
   IF (#stepNum = 6) AND "stol_final" THEN #stepNum := 2; END_IF;
END_REGION

REGION Network 11: S6 - Vrata zatvorena - spremno za okret
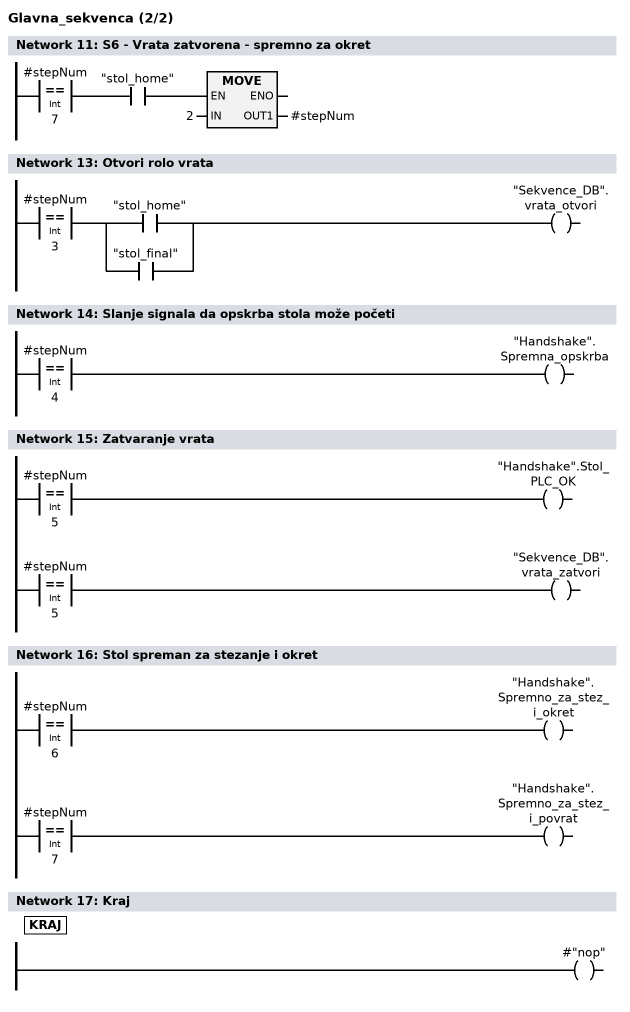
   RUNG wire#powerrail
      { S7_Templates := "SrcType := Int" } EQ_Contact(in1 := #stepNum, in2 := 7)
      Contact( "stol_home" )
      Move(in := 2, out1 => #stepNum)
   END_RUNG
   // the same network as SCL:
   IF (#stepNum = 7) AND "stol_home" THEN #stepNum := 2; END_IF;
END_REGION

REGION Network 12: RADNJE
END_REGION

REGION Network 13: Otvori rolo vrata
   RUNG wire#powerrail
      { S7_Templates := "SrcType := Int" } EQ_Contact(in1 := #stepNum, in2 := 3)
      wire#w1
      Contact( "stol_home" )
      wire#w2
      Coil( "Sekvence_DB".vrata_otvori )
   END_RUNG
   RUNG wire#w1
      Contact( "stol_final" )
   END_RUNG wire#w2
   // the same network as SCL:
   "Sekvence_DB".vrata_otvori := (#stepNum = 3) AND ("stol_home" OR "stol_final");
END_REGION

REGION Network 14: Slanje signala da opskrba stola može početi
   RUNG wire#powerrail
      { S7_Templates := "SrcType := Int" } EQ_Contact(in1 := #stepNum, in2 := 4)
      Coil( "Handshake".Spremna_opskrba )
   END_RUNG
   // the same network as SCL:
   "Handshake".Spremna_opskrba := #stepNum = 4;
END_REGION

REGION Network 15: Zatvaranje vrata
   RUNG wire#powerrail
      { S7_Templates := "SrcType := Int" } EQ_Contact(in1 := #stepNum, in2 := 5)
      Coil( "Handshake".Stol_PLC_OK )
   END_RUNG
   RUNG wire#powerrail
      { S7_Templates := "SrcType := Int" } EQ_Contact(in1 := #stepNum, in2 := 5)
      Coil( "Sekvence_DB".vrata_zatvori )
   END_RUNG
   // the same network as SCL:
   "Handshake".Stol_PLC_OK := #stepNum = 5;
   "Sekvence_DB".vrata_zatvori := #stepNum = 5;
END_REGION

REGION Network 16: Stol spreman za stezanje i okret
   RUNG wire#powerrail
      { S7_Templates := "SrcType := Int" } EQ_Contact(in1 := #stepNum, in2 := 6)
      Coil( "Handshake".Spremno_za_stez_i_okret )
   END_RUNG
   RUNG wire#powerrail
      { S7_Templates := "SrcType := Int" } EQ_Contact(in1 := #stepNum, in2 := 7)
      Coil( "Handshake".Spremno_za_stez_i_povrat )
   END_RUNG
   // the same network as SCL:
   "Handshake".Spremno_za_stez_i_okret := #stepNum = 6;
   "Handshake".Spremno_za_stez_i_povrat := #stepNum = 7;
END_REGION

REGION Network 17: Kraj
   Label( KRAJ )
   RUNG wire#powerrail
      Coil( #"nop" )
   END_RUNG
   // the same network as SCL:
   KRAJ:
   #"nop" := TRUE;
END_REGION
END_FUNCTION_BLOCK

FUNCTION_BLOCK "Robot_sekvenca"   // FB5, LAD
{ S7_Optimized_Access := 'TRUE' }
VERSION : 0.1
   VAR_INPUT
      inicijalizacija : Bool;
   END_VAR
   VAR
      bit_na_brid : Array[0..2] of Bool;
      stepNum : Int;
      stepNumPrev : Int;
   END_VAR
   VAR_TEMP
      "nop" : Bool;
   END_VAR
BEGIN

REGION Network 1: Inicijalizacija sekvence
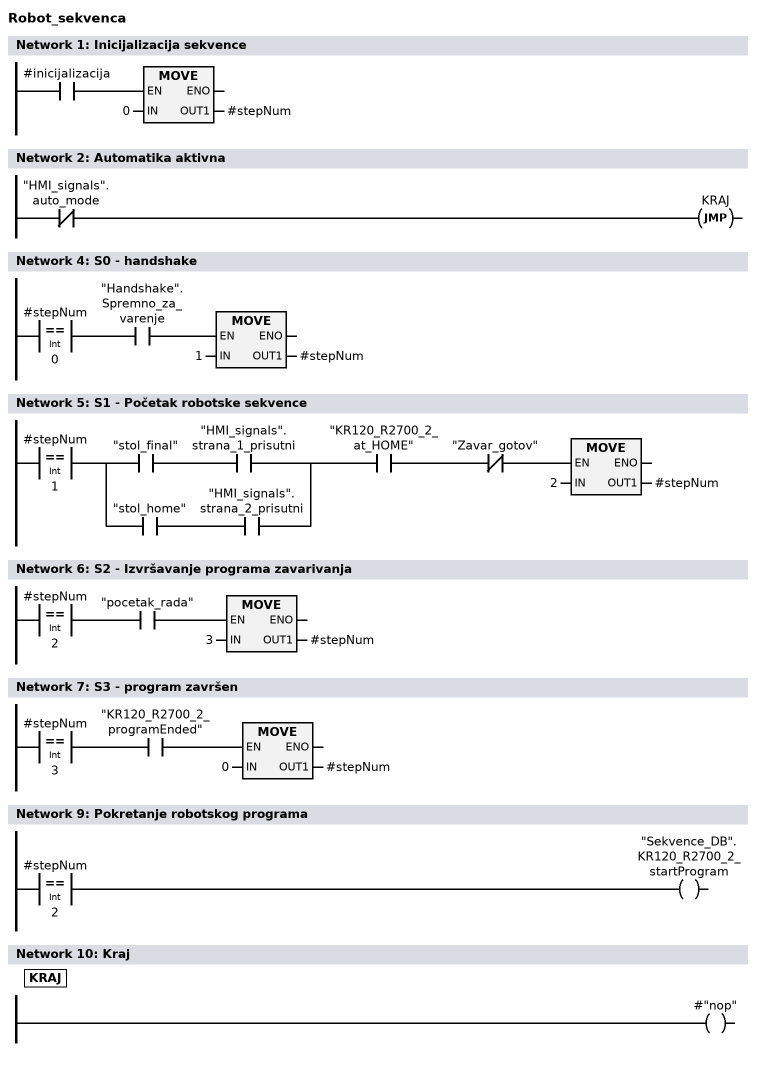
   RUNG wire#powerrail
      Contact( #inicijalizacija )
      Move(in := 0, out1 => #stepNum)
   END_RUNG
   // the same network as SCL:
   IF #inicijalizacija THEN #stepNum := 0; END_IF;
END_REGION

REGION Network 2: Automatika aktivna
   RUNG wire#powerrail
      I_Contact( "HMI_signals".auto_mode )
      JumpCoil( KRAJ )
   END_RUNG
   // the same network as SCL:
   IF NOT "HMI_signals".auto_mode THEN GOTO KRAJ; END_IF;
END_REGION

REGION Network 3: KORACI
END_REGION

REGION Network 4: S0 - handshake
   RUNG wire#powerrail
      { S7_Templates := "SrcType := Int" } EQ_Contact(in1 := #stepNum, in2 := 0)
      Contact( "Handshake".Spremno_za_varenje )
      Move(in := 1, out1 => #stepNum)
   END_RUNG
   // the same network as SCL:
   IF (#stepNum = 0) AND "Handshake".Spremno_za_varenje THEN #stepNum := 1; END_IF;
END_REGION

REGION Network 5: S1 - Početak robotske sekvence
   RUNG wire#powerrail
      { S7_Templates := "SrcType := Int" } EQ_Contact(in1 := #stepNum, in2 := 1)
      wire#w1
      Contact( "stol_final" )
      Contact( "HMI_signals".strana_1_prisutni )
      wire#w2
      Contact( "KR120_R2700_2_at_HOME" )
      I_Contact( "Zavar_gotov" )
      Move(in := 2, out1 => #stepNum)
   END_RUNG
   RUNG wire#w1
      Contact( "stol_home" )
      Contact( "HMI_signals".strana_2_prisutni )
   END_RUNG wire#w2
   // the same network as SCL:
   IF (#stepNum = 1) AND (("stol_final" AND "HMI_signals".strana_1_prisutni) OR ("stol_home" AND "HMI_signals".strana_2_prisutni)) AND "KR120_R2700_2_at_HOME" AND NOT "Zavar_gotov" THEN
       #stepNum := 2;
   END_IF;
END_REGION

REGION Network 6: S2 - Izvršavanje programa zavarivanja
   RUNG wire#powerrail
      { S7_Templates := "SrcType := Int" } EQ_Contact(in1 := #stepNum, in2 := 2)
      Contact( "pocetak_rada" )
      Move(in := 3, out1 => #stepNum)
   END_RUNG
   // the same network as SCL:
   IF (#stepNum = 2) AND "pocetak_rada" THEN #stepNum := 3; END_IF;
END_REGION

REGION Network 7: S3 - program završen
   RUNG wire#powerrail
      { S7_Templates := "SrcType := Int" } EQ_Contact(in1 := #stepNum, in2 := 3)
      Contact( "KR120_R2700_2_programEnded" )
      Move(in := 0, out1 => #stepNum)
   END_RUNG
   // the same network as SCL:
   IF (#stepNum = 3) AND "KR120_R2700_2_programEnded" THEN #stepNum := 0; END_IF;
END_REGION

REGION Network 8: RADNJE
END_REGION

REGION Network 9: Pokretanje robotskog programa
   RUNG wire#powerrail
      { S7_Templates := "SrcType := Int" } EQ_Contact(in1 := #stepNum, in2 := 2)
      Coil( "Sekvence_DB".KR120_R2700_2_startProgram )
   END_RUNG
   // the same network as SCL:
   "Sekvence_DB".KR120_R2700_2_startProgram := #stepNum = 2;
END_REGION

REGION Network 10: Kraj
   Label( KRAJ )
   RUNG wire#powerrail
      Coil( #"nop" )
   END_RUNG
   // the same network as SCL:
   KRAJ:
   #"nop" := TRUE;
END_REGION
END_FUNCTION_BLOCK

// folder: Senzori

FUNCTION_BLOCK "Senzori_prog"   // FB2, LAD
{ S7_Optimized_Access := 'TRUE' }
VERSION : 0.1
BEGIN

REGION Network 1: Senzori od stezaljka
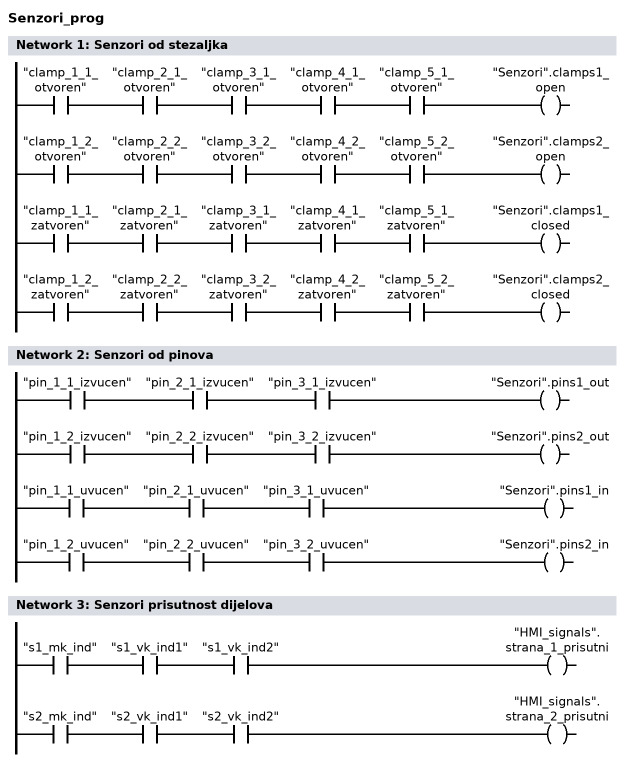
   RUNG wire#powerrail
      Contact( "clamp_1_1_otvoren" )
      Contact( "clamp_2_1_otvoren" )
      Contact( "clamp_3_1_otvoren" )
      Contact( "clamp_4_1_otvoren" )
      Contact( "clamp_5_1_otvoren" )
      Coil( "Senzori".clamps1_open )
   END_RUNG
   RUNG wire#powerrail
      Contact( "clamp_1_2_otvoren" )
      Contact( "clamp_2_2_otvoren" )
      Contact( "clamp_3_2_otvoren" )
      Contact( "clamp_4_2_otvoren" )
      Contact( "clamp_5_2_otvoren" )
      Coil( "Senzori".clamps2_open )
   END_RUNG
   RUNG wire#powerrail
      Contact( "clamp_1_1_zatvoren" )
      Contact( "clamp_2_1_zatvoren" )
      Contact( "clamp_3_1_zatvoren" )
      Contact( "clamp_4_1_zatvoren" )
      Contact( "clamp_5_1_zatvoren" )
      Coil( "Senzori".clamps1_closed )
   END_RUNG
   RUNG wire#powerrail
      Contact( "clamp_1_2_zatvoren" )
      Contact( "clamp_2_2_zatvoren" )
      Contact( "clamp_3_2_zatvoren" )
      Contact( "clamp_4_2_zatvoren" )
      Contact( "clamp_5_2_zatvoren" )
      Coil( "Senzori".clamps2_closed )
   END_RUNG
   // the same network as SCL:
   "Senzori".clamps1_open := "clamp_1_1_otvoren" AND "clamp_2_1_otvoren" AND "clamp_3_1_otvoren" AND "clamp_4_1_otvoren" AND "clamp_5_1_otvoren";
   "Senzori".clamps2_open := "clamp_1_2_otvoren" AND "clamp_2_2_otvoren" AND "clamp_3_2_otvoren" AND "clamp_4_2_otvoren" AND "clamp_5_2_otvoren";
   "Senzori".clamps1_closed := "clamp_1_1_zatvoren" AND "clamp_2_1_zatvoren" AND "clamp_3_1_zatvoren" AND "clamp_4_1_zatvoren" AND "clamp_5_1_zatvoren";
   "Senzori".clamps2_closed := "clamp_1_2_zatvoren" AND "clamp_2_2_zatvoren" AND "clamp_3_2_zatvoren" AND "clamp_4_2_zatvoren" AND "clamp_5_2_zatvoren";
END_REGION

REGION Network 2: Senzori od pinova
   RUNG wire#powerrail
      Contact( "pin_1_1_izvucen" )
      Contact( "pin_2_1_izvucen" )
      Contact( "pin_3_1_izvucen" )
      Coil( "Senzori".pins1_out )
   END_RUNG
   RUNG wire#powerrail
      Contact( "pin_1_2_izvucen" )
      Contact( "pin_2_2_izvucen" )
      Contact( "pin_3_2_izvucen" )
      Coil( "Senzori".pins2_out )
   END_RUNG
   RUNG wire#powerrail
      Contact( "pin_1_1_uvucen" )
      Contact( "pin_2_1_uvucen" )
      Contact( "pin_3_1_uvucen" )
      Coil( "Senzori".pins1_in )
   END_RUNG
   RUNG wire#powerrail
      Contact( "pin_1_2_uvucen" )
      Contact( "pin_2_2_uvucen" )
      Contact( "pin_3_2_uvucen" )
      Coil( "Senzori".pins2_in )
   END_RUNG
   // the same network as SCL:
   "Senzori".pins1_out := "pin_1_1_izvucen" AND "pin_2_1_izvucen" AND "pin_3_1_izvucen";
   "Senzori".pins2_out := "pin_1_2_izvucen" AND "pin_2_2_izvucen" AND "pin_3_2_izvucen";
   "Senzori".pins1_in := "pin_1_1_uvucen" AND "pin_2_1_uvucen" AND "pin_3_1_uvucen";
   "Senzori".pins2_in := "pin_1_2_uvucen" AND "pin_2_2_uvucen" AND "pin_3_2_uvucen";
END_REGION

REGION Network 3: Senzori prisutnost dijelova
   RUNG wire#powerrail
      Contact( "s1_mk_ind" )
      Contact( "s1_vk_ind1" )
      Contact( "s1_vk_ind2" )
      Coil( "HMI_signals".strana_1_prisutni )
   END_RUNG
   RUNG wire#powerrail
      Contact( "s2_mk_ind" )
      Contact( "s2_vk_ind1" )
      Contact( "s2_vk_ind2" )
      Coil( "HMI_signals".strana_2_prisutni )
   END_RUNG
   // the same network as SCL:
   "HMI_signals".strana_1_prisutni := "s1_mk_ind" AND "s1_vk_ind1" AND "s1_vk_ind2";
   "HMI_signals".strana_2_prisutni := "s2_mk_ind" AND "s2_vk_ind1" AND "s2_vk_ind2";
END_REGION
END_FUNCTION_BLOCK

(* ===== HMI "HMI_RT_1" =====
system functions are stored by id; their names below are inferred from use
connection "HMI_Connection_1": ETHERNET, SMART_S7_1500_OMS

HMI tags "Default tag table"
   "Tag_ScreenNumber" : UInt, internal
   "Start" : Bool = PLC pom_bits.start_auto, 1 s
   "HMI_signals_robot_start" : Bool = PLC HMI_signals.robot_start, 1 s
   "HMI_signals_robot_stop" : Bool = PLC HMI_signals.robot_stop, 1 s
   "HMI_signals_set_ventil1_ukljuci" : Bool = PLC HMI_signals.set_ventil1_ukljuci, 1 s
   "HMI_signals_set_ventil1_iskljuci" : Bool = PLC HMI_signals.set_ventil1_iskljuci, 1 s
   "HMI_signals_set_ventil2_ukljuci" : Bool = PLC HMI_signals.set_ventil2_ukljuci, 1 s
   "HMI_signals_set_ventil2_iskljuci" : Bool = PLC HMI_signals.set_ventil2_iskljuci, 1 s
   "HMI_signals_setup_mode" : Bool = PLC HMI_signals.setup_mode, 1 s
   "HMI_signals_robot_em_stop" : Bool = PLC HMI_signals.robot_em_stop, 1 s
   "HMI_signals_set_okret" : Bool = PLC HMI_signals.set_okret, 1 s
   "ventil_1_iskljuci" : Bool = PLC ventil_1_iskljuci AT %Q0.2, 1 s
   "HMI_signals_set_povratak" : Bool = PLC HMI_signals.set_povratak, 1 s
   "stol_home" : Bool = PLC stol_home AT %I4.0, 1 s
   "stol_final" : Bool = PLC stol_final AT %I4.1, 1 s
   "EstopOK" : Bool = PLC EstopOK AT %M3.0, 1 s
   "clamp_2_1_otvoren" : Bool = PLC clamp_2_1_otvoren AT %I0.3, 1 s
   "clamp_1_1_otvoren" : Bool = PLC clamp_1_1_otvoren AT %I0.1, 1 s
   "clamp_3_1_otvoren" : Bool = PLC clamp_3_1_otvoren AT %I0.5, 1 s
   "clamp_4_1_otvoren" : Bool = PLC clamp_4_1_otvoren AT %I0.7, 1 s
   "clamp_5_1_otvoren" : Bool = PLC clamp_5_1_otvoren AT %I1.1, 1 s
   "pin_1_1_izvucen" : Bool = PLC pin_1_1_izvucen AT %I2.5, 1 s
   "pin_2_1_izvucen" : Bool = PLC pin_2_1_izvucen AT %I2.7, 1 s
   "pin_3_1_izvucen" : Bool = PLC pin_3_1_izvucen AT %I3.1, 1 s
   "HMI_signals_set_ventil1_pin_ukljuci" : Bool = PLC HMI_signals.set_ventil1_pin_ukljuci, 1 s
   "HMI_signals_set_ventil1_pin_iskljuci" : Bool = PLC HMI_signals.set_ventil1_pin_iskljuci, 1 s
   "clamp_2_1_zatvoren" : Bool = PLC clamp_2_1_zatvoren AT %I0.2, 1 s
   "clamp_1_1_zatvoren" : Bool = PLC clamp_1_1_zatvoren AT %I0.0, 1 s
   "clamp_3_1_zatvoren" : Bool = PLC clamp_3_1_zatvoren AT %I0.4, 1 s
   "clamp_4_1_zatvoren" : Bool = PLC clamp_4_1_zatvoren AT %I0.6, 1 s
   "clamp_5_1_zatvoren" : Bool = PLC clamp_5_1_zatvoren AT %I1.0, 1 s
   "s1_vd_prisutan" : Bool = PLC s1_vd_prisutan AT %I4.3, 1 s
   "s1_md_prisutan" : Bool = PLC s1_md_prisutan AT %I4.2, 1 s
   "HMI_signals_s1_md_prisutan" : Bool = PLC HMI_signals.s1_md_prisutan, 1 s
   "HMI_signals_set_s1_md_stvori" : Bool = PLC HMI_signals.set_s1_md_stvori, 1 s
   "HMI_signals_set_s1_md_unisti" : Bool = PLC HMI_signals.set_s1_md_unisti, 1 s
   "Okvir_manji_unisti_start" : Bool = PLC Okvir_manji_unisti_start AT %Q3.3, 1 s
   "HMI_signals_set_s1_vd_stvori" : Bool = PLC HMI_signals.set_s1_vd_stvori, 1 s
   "Okvir_veci_unisti_start" : Bool = PLC Okvir_veci_unisti_start AT %Q3.5, 1 s
   "proximity_sensor" : Bool = PLC s1_vk_ind1 AT %I5.4, 1 s
   "s1_vk_ind2" : Bool = PLC s1_vk_ind2 AT %I5.5, 1 s
   "s1_mk_ind" : Bool = PLC s1_mk_ind AT %I5.6, 1 s
   "HMI_signals_set_zavareni" : Bool = PLC HMI_signals.set_zavareni, 1 s
   "Zavareno_unisti_start" : Bool = PLC Zavareno_unisti_start AT %Q3.7, 1 s
   "HMI_signals_prog_zavar" : Bool = PLC HMI_signals.prog_zavar, 1 s
   "HMI_signals_prog_brusenje" : Bool = PLC HMI_signals.prog_brusenje, 1 s
   "KR120_R2700_2_mirrorProgramNumber" : Byte = PLC KR120_R2700_2_mirrorProgramNumber AT %IB6, 1 s
   "handshake_test_out" : Bool = PLC handshake_test_out AT %Q4.0, 1 s
   "handshake_test_in" : Bool = PLC pocetak_rada AT %I7.1, 1 s
   "HMI_signals_auto_mode" : Bool = PLC HMI_signals.auto_mode, 1 s
   "pom_bits_automatika_aktivna" : Bool = PLC pom_bits.automatika_aktivna, 1 s
   "HMI_signals_set_vrata_otvori" : Bool = PLC HMI_signals.set_vrata_otvori, 1 s
   "HMI_signals_set_vrata_zatvori" : Bool = PLC HMI_signals.set_vrata_zatvori, 1 s
   "HMI_signals_sek_stol_res" : Bool = PLC HMI_signals.sek_stol_res, 1 s
   "HMI_signals_sek_glav_res" : Bool = PLC HMI_signals.sek_glav_res, 1 s
   "bijelo" : Bool = PLC bijelo AT %M1.1, 1 s
   "HMI_signals_set_zavareni_2" : Bool = PLC HMI_signals.set_zavareni_2, 1 s
   "Zavareno_unisti_2_start" : Bool = PLC Zavareno_unisti_2_start AT %Q7.5, 1 s
   "HMI_signals_set_s1_md_stvori_2" : Bool = PLC HMI_signals.set_s1_md_stvori_2, 1 s
   "HMI_signals_set_s1_vd_stvori_2" : Bool = PLC HMI_signals.set_s1_vd_stvori_2, 1 s
   "Okvir_manji_unisti_2_start" : Bool = PLC Okvir_manji_unisti_2_start AT %Q7.6, 1 s
   "Okvir_veci_unisti_2_start" : Bool = PLC Okvir_veci_unisti_2_start AT %Q7.4, 1 s
   "HMI_signals_set_unisti_zavarene" : Bool = PLC HMI_signals.set_unisti_zavarene, 1 s
   "HMI_signals_set_unisti_zavarene_2" : Bool = PLC HMI_signals.set_unisti_zavarene_2, 1 s
   "s2_mk_ind" : Bool = PLC s2_mk_ind AT %I9.2, 1 s
   "s2_vk_ind1" : Bool = PLC s2_vk_ind1 AT %I9.0, 1 s
   "s2_vk_ind2" : Bool = PLC s2_vk_ind2 AT %I9.1, 1 s
   "lock_otv" : Bool = PLC lock_otv AT %Q4.2, 1 s
   "lock_zat" : Bool = PLC lock_zat AT %Q4.1, 1 s
   "zeleno_svjetlo" : Bool = PLC zeleno_svjetlo AT %I5.3, 1 s
   "zuto_svjetlo" : Bool = PLC zuto_svjetlo AT %I7.6, 1 s
   "crveno_svjetlo" : Bool = PLC crveno_svjetlo AT %I7.7, 1 s
   "HMI_signals_sek_rob_res" : Bool = PLC HMI_signals.sek_rob_res, 1 s
   "HMI_signals_set_zrak" : Bool = PLC HMI_signals.set_zrak, 1 s
   "HMI_signals_reset_zrak" : Bool = PLC HMI_signals.reset_zrak, 1 s
   "pin_1_2_izvucen" : Bool = PLC pin_1_2_izvucen AT %I3.3, 1 s
   "pin_2_2_uvucen" : Bool = PLC pin_2_2_uvucen AT %I3.4, 1 s
   "pin_3_2_izvucen" : Bool = PLC pin_3_2_izvucen AT %I3.7, 1 s
   "HMI_signals_set_ventil2_pin_ukljuci" : Bool = PLC HMI_signals.set_ventil2_pin_ukljuci, 1 s
   "clamp_1_2_otvoren" : Bool = PLC clamp_1_2_otvoren AT %I1.3, 1 s
   "clamp_2_2_otvoren" : Bool = PLC clamp_2_2_otvoren AT %I1.5, 1 s
   "clamp_3_2_otvoren" : Bool = PLC clamp_3_2_otvoren AT %I1.7, 1 s
   "clamp_4_2_otvoren" : Bool = PLC clamp_4_2_otvoren AT %I2.1, 1 s
   "clamp_5_2_otvoren" : Bool = PLC clamp_5_2_otvoren AT %I2.3, 1 s
   "HMI_signals_zrak_u_sustavu" : Bool = PLC HMI_signals.zrak_u_sustavu, 1 s
   "clamp_1_2_zatvoren" : Bool = PLC clamp_1_2_zatvoren AT %I1.2, 1 s
   "clamp_2_2_zatvoren" : Bool = PLC clamp_2_2_zatvoren AT %I1.4, 1 s
   "clamp_3_2_zatvoren" : Bool = PLC clamp_3_2_zatvoren AT %I1.6, 1 s
   "clamp_4_2_zatvoren" : Bool = PLC clamp_4_2_zatvoren AT %I2.0, 1 s
   "clamp_5_2_zatvoren" : Bool = PLC clamp_5_2_zatvoren AT %I2.2, 1 s
   "HMI_signals_Estop" : Bool = PLC HMI_signals.Estop, 1 s
   "HMI_signals_lock_otv" : Bool = PLC HMI_signals.lock_otv, 1 s
   "HMI_signals_lock_zat" : Bool = PLC HMI_signals.lock_zat, 1 s

Template "Template" 800x480
   DateTimeField "HmiScreenItemData" at 689,28 size 105x25
   DateTimeField "HmiScreenItemData_1" at 689,6 size 105x25
   GraphicView "Graphic view_1" at 0,5 size 122x55; Picture "fsb_logo_1"
   GraphicView "Graphic view_2" at 242,9 size 162x44; Picture "logo_atinel"
   Button "Button_7" at 29,410 size 116x48; TextOff 'Početna'; TextOn 'Start'
      on Click: ActivateScreen("Glavni_ekran", 0)
   TextField "Text field_3" at 605,402 size 131x25; Text 'Zrak u sustavu'
   TextField "Text field_2" at 607,435 size 127x25; Text 'Isklop u nuždi'
   Circle "Circle_1" at 749,398 size 32x32
      Appearance <- "HMI_signals_zrak_u_sustavu"
   Circle "Circle_2" at 749,433 size 32x32
      Appearance <- "HMI_signals_Estop"
   GraphicView "Template_Graphic view_1" at 122,0 size 120x60; Picture "crta_logo"
   TextField "Text field_1" at 561,18 size 60x25; Text 'SETUP'
      Visibility <- "HMI_signals_setup_mode"
   TextField "Text field_4" at 562,18 size 53x25; Text 'AUTO'
      Visibility <- "pom_bits_automatika_aktivna"
   TextField "Text field_5" at 449,18 size 102x25; Text 'Način rada:'
   Button "Button_3" at 716,75 size 64x57; TextOff 'Reset'
      on Press: SetBit("bijelo")
      on Release: ResetBit("bijelo")

screen "Glavni_ekran" 800x480, template "Template_pocetna"
   Button "Button_7" at 464,220 size 200x80; TextOff 'SETUP'
      on Click: ActivateScreen("Setup_mode", 0)
      Appearance <- "HMI_signals_setup_mode"
   Button "Button_1" at 165,220 size 200x80; TextOff 'AUTO'
      on Click: SetBit("HMI_signals_auto_mode"); ResetBit("HMI_signals_setup_mode")
      Appearance <- "pom_bits_automatika_aktivna"
   TextField "Text field_1" at 307,110 size 177x43; Text 'Način rada'
   Button "Button_2" at 209,322 size 125x57; TextOff 'Pokreni'
      on Press: SetBit("Start")
      on Release: ResetBit("Start")
      Visibility <- "HMI_signals_auto_mode"
   Button "Button_3" at 36,81 size 64x57; TextOff 'Reset'
      on Press: SetBit("bijelo")
      on Release: ResetBit("bijelo")
   Rectangle "Rectangle_1" at 701,162 size 96x48
      Appearance <- "zeleno_svjetlo"
   Rectangle "Rectangle_2" at 701,64 size 96x48
      Appearance <- "crveno_svjetlo"
   Rectangle "Rectangle_3" at 701,113 size 96x48
      Appearance <- "zuto_svjetlo"

screen "Setup_mode" 800x480, template "Template"
   TextField "Text field_1" at 302,75 size 196x43; Text 'Setup mode'
   Switch "Switch_1" at 30,74 size 208x49; CaptionText 'Switch'; TextOff 'ISKLJUČEN'; TextOn 'UKLJUČEN'
      on SwitchOn: SetBit("HMI_signals_setup_mode"); ResetBit("HMI_signals_auto_mode")
      on SwitchOff: ResetBit("HMI_signals_setup_mode")
      ProcessValue <- "HMI_signals_setup_mode"
   Button "Button_1" at 59,166 size 180x55; TextOff 'Okretni stol'
      on Click: ActivateScreen("Okretni_stol", 0)
   Button "Button_2" at 59,312 size 180x55; TextOff 'Robot'
      on Click: ActivateScreen("Robot", 0)
   Button "Button_3" at 57,238 size 180x55; TextOff 'Vrata'
      on Click: ActivateScreen("Vrata", 0)
   Button "Button_4" at 373,208 size 87x28; TextOff 'Sek_res'
      on Press: SetBit("HMI_signals_sek_stol_res")
      on Release: ResetBit("HMI_signals_sek_stol_res")
   Button "Button_5" at 495,207 size 87x28; TextOff 'Sek_res'
      on Press: SetBit("HMI_signals_sek_glav_res")
      on Release: ResetBit("HMI_signals_sek_glav_res")
   Button "Button_6" at 613,207 size 87x28; TextOff 'Sek_res'
      on Press: SetBit("HMI_signals_sek_rob_res")
      on Release: ResetBit("HMI_signals_sek_stol_res")
   TextField "Text field_2" at 473,136 size 124x34; Text 'Sekvence'
   TextField "Text field_3" at 375,175 size 78x29; Text 'Glavna'
   TextField "Text field_4" at 473,175 size 128x29; Text 'Okretni stol'
   TextField "Text field_5" at 621,176 size 68x29; Text 'Robot'
   TextField "Text field_6" at 311,275 size 177x32; Text 'Zrak u sustavu'
   Button "Button_7" at 294,325 size 101x42; TextOff 'Uključi'; TextOn 'Pokreni'
      on Press: SetBit("HMI_signals_set_zrak")
      on Release: ResetBit("HMI_signals_set_zrak")
   Button "Button_8" at 407,325 size 101x42; TextOff 'Isključi'; TextOn 'Pokreni'
      on Press: SetBit("HMI_signals_reset_zrak")
      on Release: ResetBit("HMI_signals_reset_zrak")
   TextField "Text field_7" at 568,275 size 169x32; Text 'Isklop u nuždi'
   Switch "Switch_2" at 568,322 size 169x45; CaptionText 'Switch'; TextOff 'OFF'; TextOn 'ON'
      on SwitchOn: SetBit("HMI_signals_Estop")
      on SwitchOff: ResetBit("HMI_signals_Estop")
      ProcessValue <- "HMI_signals_Estop"

screen "Okretni_stol" 800x480, template "Template"
   Button "Button_9" at 68,184 size 140x60; TextOff 'Okret'; TextOn 'Natrag'
      on Press: SetBit("HMI_signals_set_okret")
      on Release: ResetBit("HMI_signals_set_okret")
   Button "Button_10" at 68,265 size 140x60; TextOff 'Povratak'; TextOn 'Natrag'
      on Press: SetBit("HMI_signals_set_povratak")
      on Release: ResetBit("HMI_signals_set_povratak")
   TextField "Text field_1" at 304,79 size 193x43; Text 'Okretni stol'
   TextField "Text field_2" at 262,235 size 81x27; Text 'Početna'
   TextField "Text field_3" at 394,235 size 86x27; Text 'Konačna'
   Circle "Circle_1" at 281,268 size 48x48
      Appearance <- "stol_home"
   Circle "Circle_2" at 415,268 size 48x48
      Appearance <- "stol_final"
   Button "Button_3" at 549,196 size 113x47; TextOff 'Strana 1'
      on Click: ActivateScreen("Strana_1", 0)
   Button "Button_4" at 549,262 size 113x47; TextOff 'Strana 2'
      on Click: ActivateScreen("Strana_2", 0)
   TextField "Text field_5" at 286,186 size 158x32; Text 'Pozicija stola'
   TextField "Text field_6" at 526,132 size 152x54; Text 'Dijelovi za pozicioniranje'
   Button "Button_7" at 185,410 size 116x48; TextOff 'Natrag'; TextOn 'Start'
      on Click: function_efd93a16()
   Button "Button_1" at 533,330 size 151x53; TextOff 'Radni komadi'
      on Click: ActivateScreen("Radni_komadi", 0)

screen "Strana_1" 800x480, template "Template"
   GraphicView "Graphic view_1" at 185,111 size 431x294; Picture "INV_strana1"
   Button "Button_2" at 49,143 size 104x33; TextOff 'Stegni'; TextOn 'Uključi'
      on Press: SetBit("HMI_signals_set_ventil1_ukljuci")
      on Release: ResetBit("HMI_signals_set_ventil1_ukljuci")
   Button "Button_4" at 49,195 size 104x33; TextOff 'Otpusti'; TextOn 'Start'
      on Press: SetBit("HMI_signals_set_ventil1_iskljuci")
      on Release: ResetBit("HMI_signals_set_ventil1_iskljuci")
   TextField "Text field_1" at 329,67 size 139x43; Text 'Strana 1'
   TextField "Text field_2" at 55,102 size 92x27; Text 'Stezaljke'
   TextField "Text field_3" at 69,246 size 64x27; Text 'Pinovi'
   Button "Button_1" at 49,284 size 104x33; TextOff 'Izvuci'; TextOn 'Uključi'
      on Press: SetBit("HMI_signals_set_ventil1_pin_ukljuci")
      on Release: ResetBit("HMI_signals_set_ventil1_pin_ukljuci")
   Button "Button_3" at 49,336 size 104x33; TextOff 'Uvuci'; TextOn 'Start'
      on Press: SetBit("HMI_signals_set_ventil1_pin_iskljuci")
      on Release: ResetBit("HMI_signals_set_ventil1_pin_iskljuci")
   Circle "Circle_1" at 256,196 size 32x32
      Appearance <- "clamp_2_1_zatvoren"
   Circle "Circle_2" at 256,284 size 32x32
      Appearance <- "clamp_1_1_zatvoren"
   Circle "Circle_3" at 388,190 size 32x32
      Appearance <- "clamp_3_1_zatvoren"
   Circle "Circle_4" at 389,290 size 32x32
      Appearance <- "clamp_4_1_zatvoren"
   Circle "Circle_6" at 517,242 size 32x32
      Appearance <- "clamp_5_1_zatvoren"
   Circle "Circle_7" at 448,351 size 32x32
      Appearance <- "pin_3_1_izvucen"
   Circle "Circle_8" at 230,138 size 32x32
      Appearance <- "pin_1_1_izvucen"
   Circle "Circle_5" at 419,241 size 32x32
      Appearance <- "pin_2_1_izvucen"
   Button "Button_7" at 185,410 size 116x48; TextOff 'Natrag'; TextOn 'Start'
      on Click: function_efd93a16()
   TextField "Text field_4" at 660,203 size 99x27; Text 'Veći okvir'
   TextField "Text field_5" at 652,300 size 112x27; Text 'Manji okvir'
   Circle "Circle_11" at 662,240 size 44x44
      Appearance <- "proximity_sensor"
   Circle "Circle_12" at 720,240 size 44x44
      Appearance <- "s1_vk_ind2"
   Circle "Circle_9" at 690,336 size 44x44
      Appearance <- "s1_mk_ind"

screen "Strana_2" 800x480, template "Template"
   Button "Button_5" at 39,147 size 113x33; TextOff 'Stegni'; TextOn 'Start'
      on Press: SetBit("HMI_signals_set_ventil2_ukljuci")
      on Release: ResetBit("HMI_signals_set_ventil2_ukljuci")
   Button "Button_6" at 39,199 size 113x33; TextOff 'Otpusti'; TextOn 'Start'
      on Press: SetBit("HMI_signals_set_ventil2_iskljuci")
      on Release: ResetBit("HMI_signals_set_ventil2_iskljuci")
   TextField "Text field_1" at 331,67 size 139x43; Text 'Strana 2'
   GraphicView "Graphic view_1" at 185,111 size 431x294; Picture "INV_strana1"
   TextField "Text field_2" at 49,106 size 92x27; Text 'Stezaljke'
   TextField "Text field_3" at 65,251 size 64x27; Text 'Pinovi'
   Button "Button_1" at 45,289 size 104x33; TextOff 'Izvuci'; TextOn 'Uključi'
      on Press: SetBit("HMI_signals_set_ventil2_pin_ukljuci")
      on Release: ResetBit("HMI_signals_set_ventil2_pin_ukljuci")
   Button "Button_3" at 45,341 size 104x33; TextOff 'Uvuci'; TextOn 'Start'
      on Press: SetBit("HMI_signals_set_ventil2_iskljuci")
      on Release: ResetBit("HMI_signals_set_ventil2_iskljuci")
   Circle "Circle_1" at 256,196 size 32x32
      Appearance <- "clamp_1_2_zatvoren"
   Circle "Circle_2" at 256,284 size 32x32
      Appearance <- "clamp_2_2_zatvoren"
   Circle "Circle_3" at 388,190 size 32x32
      Appearance <- "clamp_3_2_zatvoren"
   Circle "Circle_4" at 389,290 size 32x32
      Appearance <- "clamp_4_2_zatvoren"
   Circle "Circle_6" at 517,242 size 32x32
      Appearance <- "clamp_5_2_zatvoren"
   Circle "Circle_7" at 448,351 size 32x32
      Appearance <- "pin_3_2_izvucen"
   Circle "Circle_8" at 230,138 size 32x32
      Appearance <- "pin_1_2_izvucen"
   Circle "Circle_5" at 419,241 size 32x32
      Appearance <- "pin_2_2_uvucen"
   Button "Button_7" at 185,410 size 116x48; TextOff 'Natrag'; TextOn 'Start'
      on Click: function_efd93a16()
   TextField "Text field_4" at 660,203 size 99x27; Text 'Veći okvir'
   TextField "Text field_5" at 652,300 size 112x27; Text 'Manji okvir'
   Circle "Circle_11" at 662,240 size 44x44
      Appearance <- "s2_vk_ind1"
   Circle "Circle_12" at 720,240 size 44x44
      Appearance <- "s2_vk_ind2"
   Circle "Circle_9" at 690,336 size 44x44
      Appearance <- "s2_mk_ind"

screen "Robot" 800x480, template "Template"
   Button "Button_1" at 158,166 size 116x48; TextOff 'Start'
      on Press: SetBit("HMI_signals_robot_start")
      on Release: ResetBit("HMI_signals_robot_start")
   Button "Button_3" at 157,293 size 116x48; TextOff 'Pause'; TextOn 'Start'
      on Press: SetBit("HMI_signals_robot_stop")
      on Release: ResetBit("HMI_signals_robot_stop")
   Button "Button_8" at 157,230 size 116x48; TextOff 'Stop'; TextOn 'Start'
      on Press: SetBit("HMI_signals_robot_em_stop")
      on Release: ResetBit("HMI_signals_robot_em_stop")
   Button "Button_7" at 185,410 size 116x48; TextOff 'Natrag'; TextOn 'Start'
      on Click: function_efd93a16()
   TextField "Text field_1" at 350,99 size 101x43; Text 'Robot'
   TextField "Text field_2" at 448,174 size 184x29; Text 'Odabir programa'
   Button "Button_2" at 405,224 size 116x48; TextOff 'Zavar'; TextOn 'Start'
      on Press: SetBit("HMI_signals_prog_zavar")
      on Release: ResetBit("HMI_signals_prog_zavar")
   Button "Button_4" at 560,223 size 116x48; TextOff 'Brušenje'; TextOn 'Start'
      on Press: SetBit("HMI_signals_prog_brusenje")
      on Release: ResetBit("HMI_signals_prog_brusenje")
   Circle "Circle_4" at 443,286 size 42x42
      Appearance <- "KR120_R2700_2_mirrorProgramNumber"
   Circle "Circle_1" at 600,287 size 42x42
      Appearance <- "KR120_R2700_2_mirrorProgramNumber"

screen "Radni_komadi" 800x480, template "Template"
   Button "Button_5" at 66,235 size 136x33; TextOff 'Stvori manji'; TextOn 'Uključi'
      on Press: SetBit("HMI_signals_set_s1_md_stvori")
      on Release: ResetBit("HMI_signals_set_s1_md_stvori")
   Button "Button_6" at 65,285 size 136x33; TextOff 'Unisti manji'; TextOn 'Uključi'
      on Press: SetBit("Okvir_manji_unisti_start")
      on Release: ResetBit("Okvir_manji_unisti_start")
   TextField "Text field_1" at 288,80 size 225x43; Text 'Radni komadi'
   Button "Button_1" at 213,235 size 136x33; TextOff 'Stvori veci'; TextOn 'Uključi'
      on Press: SetBit("HMI_signals_set_s1_vd_stvori")
      on Release: ResetBit("HMI_signals_set_s1_vd_stvori")
   Button "Button_2" at 213,285 size 136x33; TextOff 'Unisti veci'; TextOn 'Uključi'
      on Press: SetBit("Okvir_veci_unisti_start")
      on Release: ResetBit("Okvir_veci_unisti_start")
   Button "Button_7" at 185,410 size 116x48; TextOff 'Natrag'; TextOn 'Start'
      on Click: function_efd93a16()
   Circle "Circle_9" at 234,331 size 44x44
      Appearance <- "proximity_sensor"
   Circle "Circle_1" at 291,332 size 44x44
      Appearance <- "s1_vk_ind2"
   Circle "Circle_2" at 115,332 size 44x44
      Appearance <- "s1_mk_ind"
   Button "Button_3" at 65,179 size 136x33; TextOff 'Izvadi zavarene'; TextOn 'Uključi'
      on Press: SetBit("HMI_signals_set_zavareni")
      on Release: ResetBit("HMI_signals_set_zavareni")
   Button "Button_4" at 212,179 size 136x33; TextOff 'Unisti zavarene'; TextOn 'Uključi'
      on Press: SetBit("HMI_signals_set_unisti_zavarene")
      on Release: ResetBit("HMI_signals_set_unisti_zavarene")
   TextField "Text field_2" at 137,127 size 139x43; Text 'Strana 1'
   TextField "Text field_3" at 527,130 size 139x43; Text 'Strana 2'
   Button "Button_8" at 461,238 size 136x33; TextOff 'Stvori manji'; TextOn 'Uključi'
      on Press: SetBit("HMI_signals_set_s1_md_stvori_2")
      on Release: ResetBit("HMI_signals_set_s1_md_stvori_2")
   Button "Button_9" at 460,288 size 136x33; TextOff 'Unisti manji'; TextOn 'Uključi'
      on Press: SetBit("Okvir_manji_unisti_2_start")
      on Release: ResetBit("Okvir_manji_unisti_2_start")
   Button "Button_10" at 608,238 size 136x33; TextOff 'Stvori veci'; TextOn 'Uključi'
      on Press: SetBit("HMI_signals_set_s1_vd_stvori_2")
      on Release: ResetBit("HMI_signals_set_s1_vd_stvori_2")
   Button "Button_11" at 608,288 size 136x33; TextOff 'Unisti veci'; TextOn 'Uključi'
      on Press: SetBit("Okvir_veci_unisti_2_start")
      on Release: ResetBit("Okvir_veci_unisti_2_start")
   Button "Button_12" at 460,182 size 136x33; TextOff 'Izvadi zavarene'; TextOn 'Uključi'
      on Press: SetBit("HMI_signals_set_zavareni_2")
      on Release: ResetBit("HMI_signals_set_zavareni_2")
   Button "Button_13" at 607,182 size 136x33; TextOff 'Unisti zavarene'; TextOn 'Uključi'
      on Press: SetBit("HMI_signals_set_unisti_zavarene_2")
      on Release: ResetBit("HMI_signals_set_unisti_zavarene_2")
   Circle "Circle_3" at 624,337 size 44x44
      Appearance <- "s2_vk_ind1"
   Circle "Circle_4" at 681,338 size 44x44
      Appearance <- "s2_vk_ind2"
   Circle "Circle_5" at 505,338 size 44x44
      Appearance <- "s2_mk_ind"

Template "Template_pocetna" 800x480
   GraphicView "Graphic view_1" at 0,5 size 122x55; Picture "fsb_logo_1"
   GraphicView "Graphic view_2" at 242,9 size 162x44; Picture "logo_atinel"
   GraphicView "Template_Graphic view_1" at 122,0 size 120x60; Picture "crta_logo"
   DateTimeField "HmiScreenItemData" at 689,28 size 105x25
   DateTimeField "HmiScreenItemData_1" at 689,6 size 105x25
   TextField "Text field_3" at 605,402 size 131x25; Text 'Zrak u sustavu'
   TextField "Text field_2" at 607,435 size 127x25; Text 'Isklop u nuždi'
   TextField "Text field_1" at 561,18 size 60x25; Text 'SETUP'
      Visibility <- "HMI_signals_setup_mode"
   TextField "Text field_4" at 562,18 size 53x25; Text 'AUTO'
      Visibility <- "pom_bits_automatika_aktivna"
   TextField "Text field_5" at 449,18 size 102x25; Text 'Način rada:'
   Circle "Circle_1" at 749,398 size 32x32
      Appearance <- "HMI_signals_zrak_u_sustavu"
   Circle "Circle_2" at 749,433 size 32x32
      Appearance <- "HMI_signals_Estop"

screen "Vrata" 800x480, template "Template"
   TextField "Text field_1" at 120,111 size 171x43; Text 'Rolo vrata'
   TextField "Text field_2" at 451,112 size 274x43; Text 'Safety lock vrata'
   Button "Button_4" at 172,192 size 104x33; TextOff 'Otvori'; TextOn 'Start'
      on Press: SetBit("HMI_signals_set_vrata_otvori")
      on Release: ResetBit("HMI_signals_set_vrata_otvori")
   Button "Button_1" at 172,250 size 104x33; TextOff 'Zatvori'; TextOn 'Start'
      on Press: SetBit("HMI_signals_set_vrata_zatvori")
      on Release: ResetBit("HMI_signals_set_vrata_zatvori")
   Button "Button_2" at 542,192 size 104x33; TextOff 'Otvori'; TextOn 'Start'
      on Press: SetBit("HMI_signals_lock_otv")
      on Release: ResetBit("HMI_signals_lock_otv")
   Button "Button_3" at 542,250 size 104x33; TextOff 'Zatvori'; TextOn 'Start'
      on Press: SetBit("HMI_signals_lock_zat")
      on Release: ResetBit("HMI_signals_lock_zat")
*)